ABB RAPID module: Module1.mod

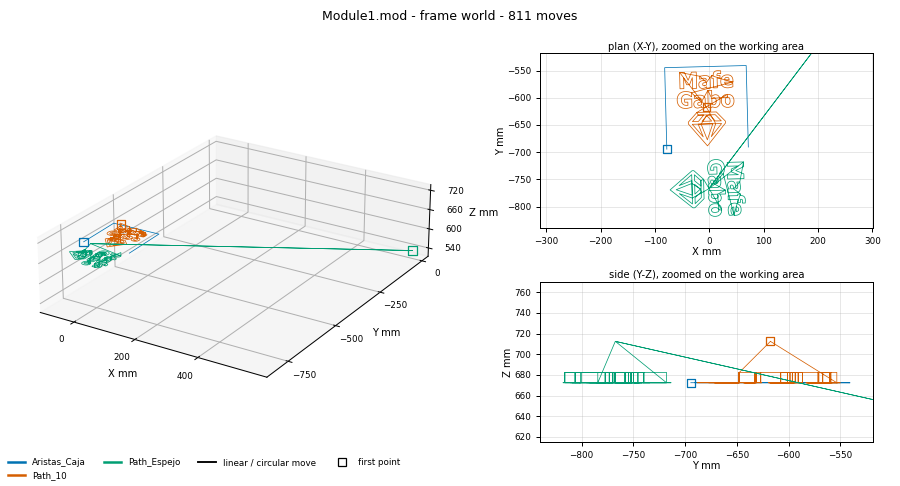
[picture p0: tool path of Module1.mod in frame world, 811 of 815 moves have a stored position in this frame; points joined in program order, loops and branches not executed]
MODULE Module1
	TASK PERS tooldata Marcador_TCP:=[TRUE,[[84.5459,-0.173285,134.639],[1,0,0,0]],[1,[1,2,3],[1,0,0,0],0,0,0]];
    !TASK PERS tooldata wcaja:=[FALSE,TRUE,"",[[-78.3768,-694.538,672.47],[0.999913,-0.00011372,0.00016022,0.0132033]],[[-74.9038,-552.314,679.445],[0.0262226,-0.999656,6.92619E-06,1.8063E-05]]];
    !TASK PERS wobjdata Caja:=[FALSE,TRUE,"",[[-250,0,346],[1,0,0,0]],[[750,75,154],[0.707106781,0,0,-0.707106781]]];
    !TASK PERS wobjdata Caja:=[FALSE,TRUE,"",[[-78.3768,-694.538,672.47],[0.999913,-0.00011372,0.00016022,0.0132033]],[[-74.9038,-552.314,679.445],[0.0262226,-0.999656,0.000006926,0.000018063]]];
    !TASK PERS wobjdata wcaja:=[FALSE,TRUE,"",[[-78.3768,-694.538,672.47],[0.999913,-0.00011372,0.00016022,0.0132033]],[[-74.9038,-552.314,679.445],[0.0262226,-0.999656,6.92619E-06,1.8063E-05]]];
    CONST robtarget Home:=[[75.173285,80.619495586,38.961602814],[0.353553391,-0.612372436,0.612372436,0.353553391],[0,0,0,0],[9E+09,9E+09,9E+09,9E+09,9E+09,9E+09]];
    CONST robtarget Target_10:=[[0,0,0],[0.353553391,0.612372436,0.612372436,-0.353553391],[0,-1,0,0],[9E+09,9E+09,9E+09,9E+09,9E+09,9E+09]];
    CONST robtarget Target_20:=[[0,150,0],[0.353553391,0.612372436,0.612372436,-0.353553391],[0,-1,0,0],[9E+09,9E+09,9E+09,9E+09,9E+09,9E+09]];
    CONST robtarget Target_30:=[[150,150,0],[0.353553391,0.612372436,0.612372436,-0.353553391],[-1,0,-1,0],[9E+09,9E+09,9E+09,9E+09,9E+09,9E+09]];
    CONST robtarget Target_40:=[[150,0,0],[0.353553391,0.612372436,0.612372436,-0.353553391],[-1,0,-1,0],[9E+09,9E+09,9E+09,9E+09,9E+09,9E+09]];
    CONST robtarget Target_50:=[[27.192,140.456999999,10],[0,0.866025404,0,-0.499999999],[0,0,0,0],[9E+09,9E+09,9E+09,9E+09,9E+09,9E+09]];
    CONST robtarget Target_60:=[[27.192,140.457,0],[0.353553391,0.612372436,0.612372436,-0.353553391],[-2,0,-1,0],[9E+09,9E+09,9E+09,9E+09,9E+09,9E+09]];
    CONST robtarget Target_70:=[[35.871,140.457,0],[0.353553391,0.612372436,0.612372436,-0.353553391],[-2,0,-1,0],[9E+09,9E+09,9E+09,9E+09,9E+09,9E+09]];
    CONST robtarget Target_80:=[[42.532,125.651,0],[0.353553391,0.612372436,0.612372436,-0.353553391],[-2,0,-1,0],[9E+09,9E+09,9E+09,9E+09,9E+09,9E+09]];
    CONST robtarget Target_90:=[[49.145,140.457,0],[0.353553391,0.612372436,0.612372436,-0.353553391],[-2,0,-1,0],[9E+09,9E+09,9E+09,9E+09,9E+09,9E+09]];
    CONST robtarget Target_100:=[[57.824,140.457,0],[0.353553391,0.612372436,0.612372436,-0.353553391],[-2,0,-1,0],[9E+09,9E+09,9E+09,9E+09,9E+09,9E+09]];
    CONST robtarget Target_110:=[[57.824,110.457,0],[0.353553391,0.612372436,0.612372436,-0.353553391],[-2,0,-1,0],[9E+09,9E+09,9E+09,9E+09,9E+09,9E+09]];
    CONST robtarget Target_120:=[[50.336,110.457,0],[0.353553391,0.612372436,0.612372436,-0.353553391],[-2,0,-1,0],[9E+09,9E+09,9E+09,9E+09,9E+09,9E+09]];
    CONST robtarget Target_130:=[[50.336,130.343,0],[0.353553391,0.612372436,0.612372436,-0.353553391],[-2,0,-1,0],[9E+09,9E+09,9E+09,9E+09,9E+09,9E+09]];
    CONST robtarget Target_140:=[[44.891,117.507,0],[0.353553391,0.612372436,0.612372436,-0.353553391],[-2,0,-1,0],[9E+09,9E+09,9E+09,9E+09,9E+09,9E+09]];
    CONST robtarget Target_150:=[[39.737,117.507,0],[0.353553391,0.612372436,0.612372436,-0.353553391],[-2,0,-1,0],[9E+09,9E+09,9E+09,9E+09,9E+09,9E+09]];
    CONST robtarget Target_160:=[[34.291,130.343,0],[0.353553391,0.612372436,0.612372436,-0.353553391],[-2,0,-1,0],[9E+09,9E+09,9E+09,9E+09,9E+09,9E+09]];
    CONST robtarget Target_170:=[[34.291,110.457,0],[0.353553391,0.612372436,0.612372436,-0.353553391],[-2,0,-1,0],[9E+09,9E+09,9E+09,9E+09,9E+09,9E+09]];
    CONST robtarget Target_180:=[[27.192,110.457,0],[0.353553391,0.612372436,0.612372436,-0.353553391],[-2,0,-1,0],[9E+09,9E+09,9E+09,9E+09,9E+09,9E+09]];
    CONST robtarget Target_190:=[[27.192,140.457,0],[0.353553391,0.612372436,0.612372436,-0.353553391],[-2,0,-1,0],[9E+09,9E+09,9E+09,9E+09,9E+09,9E+09]];
    CONST robtarget Target_200:=[[27.192,140.457,10],[0.353553391,0.612372436,0.612372436,-0.353553391],[-2,0,-1,0],[9E+09,9E+09,9E+09,9E+09,9E+09,9E+09]];
    CONST robtarget Target_210:=[[63.829,132.604,10],[0.353553391,0.612372436,0.612372436,-0.353553391],[-2,0,-1,0],[9E+09,9E+09,9E+09,9E+09,9E+09,9E+09]];
    CONST robtarget Target_220:=[[63.829,132.604,0],[0.353553391,0.612372436,0.612372436,-0.353553391],[-2,0,-1,0],[9E+09,9E+09,9E+09,9E+09,9E+09,9E+09]];
    CONST robtarget Target_230:=[[71.925,133.722,0],[0.353553391,0.612372436,0.612372436,-0.353553391],[-2,0,-1,0],[9E+09,9E+09,9E+09,9E+09,9E+09,9E+09]];
    CONST robtarget Target_240:=[[73.075,133.702,0],[0.353553391,0.612372436,0.612372436,-0.353553391],[-2,0,-1,0],[9E+09,9E+09,9E+09,9E+09,9E+09,9E+09]];
    CONST robtarget Target_250:=[[74.399,133.623,0],[0.353553391,0.612372436,0.612372436,-0.353553391],[-2,0,-1,0],[9E+09,9E+09,9E+09,9E+09,9E+09,9E+09]];
    CONST robtarget Target_260:=[[76.16,133.399,0],[0.353553391,0.612372436,0.612372436,-0.353553391],[-2,0,-1,0],[9E+09,9E+09,9E+09,9E+09,9E+09,9E+09]];
    CONST robtarget Target_270:=[[77.475,133.111,0],[0.353553391,0.612372436,0.612372436,-0.353553391],[-2,0,-1,0],[9E+09,9E+09,9E+09,9E+09,9E+09,9E+09]];
    CONST robtarget Target_280:=[[78.922,132.618,0],[0.353553391,0.612372436,0.612372436,-0.353553391],[-2,0,-1,0],[9E+09,9E+09,9E+09,9E+09,9E+09,9E+09]];
    CONST robtarget Target_290:=[[80.057,132.032,0],[0.353553391,0.612372436,0.612372436,-0.353553391],[-2,0,-1,0],[9E+09,9E+09,9E+09,9E+09,9E+09,9E+09]];
    CONST robtarget Target_300:=[[81.155,131.169,0],[0.353553391,0.612372436,0.612372436,-0.353553391],[-2,0,-1,0],[9E+09,9E+09,9E+09,9E+09,9E+09,9E+09]];
    CONST robtarget Target_310:=[[81.768,130.466,0],[0.353553391,0.612372436,0.612372436,-0.353553391],[-2,0,-1,0],[9E+09,9E+09,9E+09,9E+09,9E+09,9E+09]];
    CONST robtarget Target_320:=[[82.441,129.318,0],[0.353553391,0.612372436,0.612372436,-0.353553391],[-2,0,-1,0],[9E+09,9E+09,9E+09,9E+09,9E+09,9E+09]];
    CONST robtarget Target_330:=[[82.754,128.475,0],[0.353553391,0.612372436,0.612372436,-0.353553391],[-2,0,-1,0],[9E+09,9E+09,9E+09,9E+09,9E+09,9E+09]];
    CONST robtarget Target_340:=[[82.989,127.436,0],[0.353553391,0.612372436,0.612372436,-0.353553391],[-2,0,-1,0],[9E+09,9E+09,9E+09,9E+09,9E+09,9E+09]];
    CONST robtarget Target_350:=[[83.108,125.846,0],[0.353553391,0.612372436,0.612372436,-0.353553391],[-2,0,-1,0],[9E+09,9E+09,9E+09,9E+09,9E+09,9E+09]];
    CONST robtarget Target_360:=[[83.108,110.457,0],[0.353553391,0.612372436,0.612372436,-0.353553391],[-2,0,-1,0],[9E+09,9E+09,9E+09,9E+09,9E+09,9E+09]];
    CONST robtarget Target_370:=[[76.106,110.457,0],[0.353553391,0.612372436,0.612372436,-0.353553391],[-2,0,-1,0],[9E+09,9E+09,9E+09,9E+09,9E+09,9E+09]];
    CONST robtarget Target_380:=[[76.106,112.863,0],[0.353553391,0.612372436,0.612372436,-0.353553391],[-2,0,-1,0],[9E+09,9E+09,9E+09,9E+09,9E+09,9E+09]];
    CONST robtarget Target_390:=[[73.262,110.797,0],[0.353553391,0.612372436,0.612372436,-0.353553391],[-2,0,-1,0],[9E+09,9E+09,9E+09,9E+09,9E+09,9E+09]];
    CONST robtarget Target_400:=[[68.91,109.849,0],[0.353553391,0.612372436,0.612372436,-0.353553391],[-2,0,-1,0],[9E+09,9E+09,9E+09,9E+09,9E+09,9E+09]];
    CONST robtarget Target_410:=[[67.809,109.921,0],[0.353553391,0.612372436,0.612372436,-0.353553391],[-2,0,-1,0],[9E+09,9E+09,9E+09,9E+09,9E+09,9E+09]];
    CONST robtarget Target_420:=[[66.698,110.161,0],[0.353553391,0.612372436,0.612372436,-0.353553391],[-2,0,-1,0],[9E+09,9E+09,9E+09,9E+09,9E+09,9E+09]];
    CONST robtarget Target_430:=[[65.802,110.508,0],[0.353553391,0.612372436,0.612372436,-0.353553391],[-2,0,-1,0],[9E+09,9E+09,9E+09,9E+09,9E+09,9E+09]];
    CONST robtarget Target_440:=[[64.811,111.094,0],[0.353553391,0.612372436,0.612372436,-0.353553391],[-2,0,-1,0],[9E+09,9E+09,9E+09,9E+09,9E+09,9E+09]];
    CONST robtarget Target_450:=[[63.886,111.896,0],[0.353553391,0.612372436,0.612372436,-0.353553391],[-2,0,-1,0],[9E+09,9E+09,9E+09,9E+09,9E+09,9E+09]];
    CONST robtarget Target_460:=[[63.01,112.999,0],[0.353553391,0.612372436,0.612372436,-0.353553391],[-2,0,-1,0],[9E+09,9E+09,9E+09,9E+09,9E+09,9E+09]];
    CONST robtarget Target_470:=[[62.505,113.958,0],[0.353553391,0.612372436,0.612372436,-0.353553391],[-2,0,-1,0],[9E+09,9E+09,9E+09,9E+09,9E+09,9E+09]];
    CONST robtarget Target_480:=[[62.106,115.23,0],[0.353553391,0.612372436,0.612372436,-0.353553391],[-2,0,-1,0],[9E+09,9E+09,9E+09,9E+09,9E+09,9E+09]];
    CONST robtarget Target_490:=[[61.935,116.747,0],[0.353553391,0.612372436,0.612372436,-0.353553391],[-2,0,-1,0],[9E+09,9E+09,9E+09,9E+09,9E+09,9E+09]];
    CONST robtarget Target_500:=[[61.956,117.693,0],[0.353553391,0.612372436,0.612372436,-0.353553391],[-2,0,-1,0],[9E+09,9E+09,9E+09,9E+09,9E+09,9E+09]];
    CONST robtarget Target_510:=[[62.24,119.422,0],[0.353553391,0.612372436,0.612372436,-0.353553391],[-2,0,-1,0],[9E+09,9E+09,9E+09,9E+09,9E+09,9E+09]];
    CONST robtarget Target_520:=[[62.681,120.558,0],[0.353553391,0.612372436,0.612372436,-0.353553391],[-2,0,-1,0],[9E+09,9E+09,9E+09,9E+09,9E+09,9E+09]];
    CONST robtarget Target_530:=[[63.326,121.537,0],[0.353553391,0.612372436,0.612372436,-0.353553391],[-2,0,-1,0],[9E+09,9E+09,9E+09,9E+09,9E+09,9E+09]];
    CONST robtarget Target_540:=[[64.156,122.386,0],[0.353553391,0.612372436,0.612372436,-0.353553391],[-2,0,-1,0],[9E+09,9E+09,9E+09,9E+09,9E+09,9E+09]];
    CONST robtarget Target_550:=[[65.088,123.055,0],[0.353553391,0.612372436,0.612372436,-0.353553391],[-2,0,-1,0],[9E+09,9E+09,9E+09,9E+09,9E+09,9E+09]];
    CONST robtarget Target_560:=[[65.847,123.463,0],[0.353553391,0.612372436,0.612372436,-0.353553391],[-2,0,-1,0],[9E+09,9E+09,9E+09,9E+09,9E+09,9E+09]];
    CONST robtarget Target_570:=[[69.214,124.548,0],[0.353553391,0.612372436,0.612372436,-0.353553391],[-2,0,-1,0],[9E+09,9E+09,9E+09,9E+09,9E+09,9E+09]];
    CONST robtarget Target_580:=[[70.751,124.795,0],[0.353553391,0.612372436,0.612372436,-0.353553391],[-2,0,-1,0],[9E+09,9E+09,9E+09,9E+09,9E+09,9E+09]];
    CONST robtarget Target_590:=[[72.603,125.014,0],[0.353553391,0.612372436,0.612372436,-0.353553391],[-2,0,-1,0],[9E+09,9E+09,9E+09,9E+09,9E+09,9E+09]];
    CONST robtarget Target_600:=[[74.414,125.184,0],[0.353553391,0.612372436,0.612372436,-0.353553391],[-2,0,-1,0],[9E+09,9E+09,9E+09,9E+09,9E+09,9E+09]];
    CONST robtarget Target_610:=[[76.155,125.311,0],[0.353553391,0.612372436,0.612372436,-0.353553391],[-2,0,-1,0],[9E+09,9E+09,9E+09,9E+09,9E+09,9E+09]];
    CONST robtarget Target_620:=[[76.155,125.432,0],[0.353553391,0.612372436,0.612372436,-0.353553391],[-2,0,-1,0],[9E+09,9E+09,9E+09,9E+09,9E+09,9E+09]];
    CONST robtarget Target_630:=[[76.114,126.039,0],[0.353553391,0.612372436,0.612372436,-0.353553391],[-2,0,-1,0],[9E+09,9E+09,9E+09,9E+09,9E+09,9E+09]];
    CONST robtarget Target_640:=[[75.849,126.936,0],[0.353553391,0.612372436,0.612372436,-0.353553391],[-2,0,-1,0],[9E+09,9E+09,9E+09,9E+09,9E+09,9E+09]];
    CONST robtarget Target_650:=[[75.219,127.729,0],[0.353553391,0.612372436,0.612372436,-0.353553391],[-2,0,-1,0],[9E+09,9E+09,9E+09,9E+09,9E+09,9E+09]];
    CONST robtarget Target_660:=[[74.486,128.154,0],[0.353553391,0.612372436,0.612372436,-0.353553391],[-2,0,-1,0],[9E+09,9E+09,9E+09,9E+09,9E+09,9E+09]];
    CONST robtarget Target_670:=[[73.351,128.499,0],[0.353553391,0.612372436,0.612372436,-0.353553391],[-2,0,-1,0],[9E+09,9E+09,9E+09,9E+09,9E+09,9E+09]];
    CONST robtarget Target_680:=[[72.285,128.661,0],[0.353553391,0.612372436,0.612372436,-0.353553391],[-2,0,-1,0],[9E+09,9E+09,9E+09,9E+09,9E+09,9E+09]];
    CONST robtarget Target_690:=[[71.471,128.72,0],[0.353553391,0.612372436,0.612372436,-0.353553391],[-2,0,-1,0],[9E+09,9E+09,9E+09,9E+09,9E+09,9E+09]];
    CONST robtarget Target_700:=[[70.612,128.739,0],[0.353553391,0.612372436,0.612372436,-0.353553391],[-2,0,-1,0],[9E+09,9E+09,9E+09,9E+09,9E+09,9E+09]];
    CONST robtarget Target_710:=[[64.437,127.134,0],[0.353553391,0.612372436,0.612372436,-0.353553391],[-2,0,-1,0],[9E+09,9E+09,9E+09,9E+09,9E+09,9E+09]];
    CONST robtarget Target_720:=[[63.829,127.134,0],[0.353553391,0.612372436,0.612372436,-0.353553391],[-2,0,-1,0],[9E+09,9E+09,9E+09,9E+09,9E+09,9E+09]];
    CONST robtarget Target_730:=[[63.829,132.604,0],[0.353553391,0.612372436,0.612372436,-0.353553391],[-2,0,-1,0],[9E+09,9E+09,9E+09,9E+09,9E+09,9E+09]];
    CONST robtarget Target_740:=[[63.829,132.604,10],[0.353553391,0.612372436,0.612372436,-0.353553391],[-2,0,-1,0],[9E+09,9E+09,9E+09,9E+09,9E+09,9E+09]];
    CONST robtarget Target_750:=[[76.106,121.056,10],[0.353553391,0.612372436,0.612372436,-0.353553391],[-2,0,-1,0],[9E+09,9E+09,9E+09,9E+09,9E+09,9E+09]];
    CONST robtarget Target_760:=[[76.106,121.056,0],[0.353553391,0.612372436,0.612372436,-0.353553391],[-2,0,-1,0],[9E+09,9E+09,9E+09,9E+09,9E+09,9E+09]];
    CONST robtarget Target_770:=[[71.025,120.23,0],[0.353553391,0.612372436,0.612372436,-0.353553391],[-2,0,-1,0],[9E+09,9E+09,9E+09,9E+09,9E+09,9E+09]];
    CONST robtarget Target_780:=[[70.06,119.739,0],[0.353553391,0.612372436,0.612372436,-0.353553391],[-2,0,-1,0],[9E+09,9E+09,9E+09,9E+09,9E+09,9E+09]];
    CONST robtarget Target_790:=[[69.338,118.892,0],[0.353553391,0.612372436,0.612372436,-0.353553391],[-2,0,-1,0],[9E+09,9E+09,9E+09,9E+09,9E+09,9E+09]];
    CONST robtarget Target_800:=[[69.114,118.205,0],[0.353553391,0.612372436,0.612372436,-0.353553391],[-2,0,-1,0],[9E+09,9E+09,9E+09,9E+09,9E+09,9E+09]];
    CONST robtarget Target_810:=[[69.056,117.55,0],[0.353553391,0.612372436,0.612372436,-0.353553391],[-2,0,-1,0],[9E+09,9E+09,9E+09,9E+09,9E+09,9E+09]];
    CONST robtarget Target_820:=[[69.091,116.93,0],[0.353553391,0.612372436,0.612372436,-0.353553391],[-2,0,-1,0],[9E+09,9E+09,9E+09,9E+09,9E+09,9E+09]];
    CONST robtarget Target_830:=[[69.292,116.148,0],[0.353553391,0.612372436,0.612372436,-0.353553391],[-2,0,-1,0],[9E+09,9E+09,9E+09,9E+09,9E+09,9E+09]];
    CONST robtarget Target_840:=[[69.919,115.356,0],[0.353553391,0.612372436,0.612372436,-0.353553391],[-2,0,-1,0],[9E+09,9E+09,9E+09,9E+09,9E+09,9E+09]];
    CONST robtarget Target_850:=[[70.774,114.964,0],[0.353553391,0.612372436,0.612372436,-0.353553391],[-2,0,-1,0],[9E+09,9E+09,9E+09,9E+09,9E+09,9E+09]];
    CONST robtarget Target_860:=[[71.742,114.79,0],[0.353553391,0.612372436,0.612372436,-0.353553391],[-2,0,-1,0],[9E+09,9E+09,9E+09,9E+09,9E+09,9E+09]];
    CONST robtarget Target_870:=[[72.46,114.76,0],[0.353553391,0.612372436,0.612372436,-0.353553391],[-2,0,-1,0],[9E+09,9E+09,9E+09,9E+09,9E+09,9E+09]];
    CONST robtarget Target_880:=[[72.459,114.76,0],[0.353553391,0.612372436,0.612372436,-0.353553391],[-2,0,-1,0],[9E+09,9E+09,9E+09,9E+09,9E+09,9E+09]];
    CONST robtarget Target_890:=[[73.597,114.916,0],[0.353553391,0.612372436,0.612372436,-0.353553391],[-2,0,-1,0],[9E+09,9E+09,9E+09,9E+09,9E+09,9E+09]];
    CONST robtarget Target_900:=[[74.622,115.309,0],[0.353553391,0.612372436,0.612372436,-0.353553391],[-2,0,-1,0],[9E+09,9E+09,9E+09,9E+09,9E+09,9E+09]];
    CONST robtarget Target_910:=[[75.105,115.58,0],[0.353553391,0.612372436,0.612372436,-0.353553391],[-2,0,-1,0],[9E+09,9E+09,9E+09,9E+09,9E+09,9E+09]];
    CONST robtarget Target_920:=[[75.771,116.063,0],[0.353553391,0.612372436,0.612372436,-0.353553391],[-2,0,-1,0],[9E+09,9E+09,9E+09,9E+09,9E+09,9E+09]];
    CONST robtarget Target_930:=[[76.106,116.364,0],[0.353553391,0.612372436,0.612372436,-0.353553391],[-2,0,-1,0],[9E+09,9E+09,9E+09,9E+09,9E+09,9E+09]];
    CONST robtarget Target_940:=[[76.106,121.056,0],[0.353553391,0.612372436,0.612372436,-0.353553391],[-2,0,-1,0],[9E+09,9E+09,9E+09,9E+09,9E+09,9E+09]];
    CONST robtarget Target_950:=[[76.106,121.056,10],[0.353553391,0.612372436,0.612372436,-0.353553391],[-2,0,-1,0],[9E+09,9E+09,9E+09,9E+09,9E+09,9E+09]];
    CONST robtarget Target_960:=[[86.049,133.09,10],[0.353553391,0.612372436,0.612372436,-0.353553391],[-1,0,-1,0],[9E+09,9E+09,9E+09,9E+09,9E+09,9E+09]];
    CONST robtarget Target_970:=[[86.049,133.09,0],[0.353553391,0.612372436,0.612372436,-0.353553391],[-1,0,-1,0],[9E+09,9E+09,9E+09,9E+09,9E+09,9E+09]];
    CONST robtarget Target_980:=[[88.87,133.09,0],[0.353553391,0.612372436,0.612372436,-0.353553391],[-1,0,-1,0],[9E+09,9E+09,9E+09,9E+09,9E+09,9E+09]];
    CONST robtarget Target_990:=[[88.87,133.722,0],[0.353553391,0.612372436,0.612372436,-0.353553391],[-1,0,-1,0],[9E+09,9E+09,9E+09,9E+09,9E+09,9E+09]];
    CONST robtarget Target_1000:=[[88.943,135.17,0],[0.353553391,0.612372436,0.612372436,-0.353553391],[-1,0,-1,0],[9E+09,9E+09,9E+09,9E+09,9E+09,9E+09]];
    CONST robtarget Target_1010:=[[89.33,137.086,0],[0.353553391,0.612372436,0.612372436,-0.353553391],[-1,0,-1,0],[9E+09,9E+09,9E+09,9E+09,9E+09,9E+09]];
    CONST robtarget Target_1020:=[[90.035,138.666,0],[0.353553391,0.612372436,0.612372436,-0.353553391],[-1,0,-1,0],[9E+09,9E+09,9E+09,9E+09,9E+09,9E+09]];
    CONST robtarget Target_1030:=[[90.843,139.72,0],[0.353553391,0.612372436,0.612372436,-0.353553391],[-1,0,-1,0],[9E+09,9E+09,9E+09,9E+09,9E+09,9E+09]];
    CONST robtarget Target_1040:=[[92.423,140.908,0],[0.353553391,0.612372436,0.612372436,-0.353553391],[-1,0,-1,0],[9E+09,9E+09,9E+09,9E+09,9E+09,9E+09]];
    CONST robtarget Target_1050:=[[94.644,141.698,0],[0.353553391,0.612372436,0.612372436,-0.353553391],[-1,0,-1,0],[9E+09,9E+09,9E+09,9E+09,9E+09,9E+09]];
    CONST robtarget Target_1060:=[[96.483,141.95,0],[0.353553391,0.612372436,0.612372436,-0.353553391],[-1,-1,-1,0],[9E+09,9E+09,9E+09,9E+09,9E+09,9E+09]];
    CONST robtarget Target_1070:=[[97.646,141.988,0],[0.353553391,0.612372436,0.612372436,-0.353553391],[-1,-1,0,0],[9E+09,9E+09,9E+09,9E+09,9E+09,9E+09]];
    CONST robtarget Target_1080:=[[102.8,141.575,0],[0.353553391,0.612372436,0.612372436,-0.353553391],[-1,-1,0,0],[9E+09,9E+09,9E+09,9E+09,9E+09,9E+09]];
    CONST robtarget Target_1090:=[[102.8,136.47,0],[0.353553391,0.612372436,0.612372436,-0.353553391],[-1,-1,0,0],[9E+09,9E+09,9E+09,9E+09,9E+09,9E+09]];
    CONST robtarget Target_1100:=[[102.265,136.47,0],[0.353553391,0.612372436,0.612372436,-0.353553391],[-1,-1,0,0],[9E+09,9E+09,9E+09,9E+09,9E+09,9E+09]];
    CONST robtarget Target_1110:=[[99.372,136.98,0],[0.353553391,0.612372436,0.612372436,-0.353553391],[-1,-1,0,0],[9E+09,9E+09,9E+09,9E+09,9E+09,9E+09]];
    CONST robtarget Target_1120:=[[98.552,136.947,0],[0.353553391,0.612372436,0.612372436,-0.353553391],[-1,-1,0,0],[9E+09,9E+09,9E+09,9E+09,9E+09,9E+09]];
    CONST robtarget Target_1130:=[[97.623,136.799,0],[0.353553391,0.612372436,0.612372436,-0.353553391],[-1,-1,0,0],[9E+09,9E+09,9E+09,9E+09,9E+09,9E+09]];
    CONST robtarget Target_1140:=[[96.675,136.388,0],[0.353553391,0.612372436,0.612372436,-0.353553391],[-1,-1,0,0],[9E+09,9E+09,9E+09,9E+09,9E+09,9E+09]];
    CONST robtarget Target_1150:=[[96.077,135.652,0],[0.353553391,0.612372436,0.612372436,-0.353553391],[-1,0,-1,0],[9E+09,9E+09,9E+09,9E+09,9E+09,9E+09]];
    CONST robtarget Target_1160:=[[95.864,135.05,0],[0.353553391,0.612372436,0.612372436,-0.353553391],[-1,0,-1,0],[9E+09,9E+09,9E+09,9E+09,9E+09,9E+09]];
    CONST robtarget Target_1170:=[[95.723,134.236,0],[0.353553391,0.612372436,0.612372436,-0.353553391],[-1,0,-1,0],[9E+09,9E+09,9E+09,9E+09,9E+09,9E+09]];
    CONST robtarget Target_1180:=[[95.677,133.26,0],[0.353553391,0.612372436,0.612372436,-0.353553391],[-1,0,-1,0],[9E+09,9E+09,9E+09,9E+09,9E+09,9E+09]];
    CONST robtarget Target_1190:=[[95.677,133.09,0],[0.353553391,0.612372436,0.612372436,-0.353553391],[-1,0,-1,0],[9E+09,9E+09,9E+09,9E+09,9E+09,9E+09]];
    CONST robtarget Target_1200:=[[101.293,133.09,0],[0.353553391,0.612372436,0.612372436,-0.353553391],[-1,-1,0,0],[9E+09,9E+09,9E+09,9E+09,9E+09,9E+09]];
    CONST robtarget Target_1210:=[[101.293,128.179,0],[0.353553391,0.612372436,0.612372436,-0.353553391],[-1,-1,0,0],[9E+09,9E+09,9E+09,9E+09,9E+09,9E+09]];
    CONST robtarget Target_1220:=[[95.92,128.179,0],[0.353553391,0.612372436,0.612372436,-0.353553391],[-1,0,-1,0],[9E+09,9E+09,9E+09,9E+09,9E+09,9E+09]];
    CONST robtarget Target_1230:=[[95.92,110.457,0],[0.353553391,0.612372436,0.612372436,-0.353553391],[-1,0,-1,0],[9E+09,9E+09,9E+09,9E+09,9E+09,9E+09]];
    CONST robtarget Target_1240:=[[88.87,110.457,0],[0.353553391,0.612372436,0.612372436,-0.353553391],[-1,0,-1,0],[9E+09,9E+09,9E+09,9E+09,9E+09,9E+09]];
    CONST robtarget Target_1250:=[[88.87,128.179,0],[0.353553391,0.612372436,0.612372436,-0.353553391],[-1,0,-1,0],[9E+09,9E+09,9E+09,9E+09,9E+09,9E+09]];
    CONST robtarget Target_1260:=[[86.049,128.179,0],[0.353553391,0.612372436,0.612372436,-0.353553391],[-1,0,-1,0],[9E+09,9E+09,9E+09,9E+09,9E+09,9E+09]];
    CONST robtarget Target_1270:=[[86.049,133.09,0],[0.353553391,0.612372436,0.612372436,-0.353553391],[-1,0,-1,0],[9E+09,9E+09,9E+09,9E+09,9E+09,9E+09]];
    CONST robtarget Target_1280:=[[86.049,133.09,10],[0.353553391,0.612372436,0.612372436,-0.353553391],[-1,0,-1,0],[9E+09,9E+09,9E+09,9E+09,9E+09,9E+09]];
    CONST robtarget Target_1290:=[[109.485,124.679,10],[0.353553391,0.612372436,0.612372436,-0.353553391],[-1,-1,0,0],[9E+09,9E+09,9E+09,9E+09,9E+09,9E+09]];
    CONST robtarget Target_1300:=[[109.485,124.679,0],[0.353553391,0.612372436,0.612372436,-0.353553391],[-1,-1,0,0],[9E+09,9E+09,9E+09,9E+09,9E+09,9E+09]];
    CONST robtarget Target_1310:=[[109.701,126.061,0],[0.353553391,0.612372436,0.612372436,-0.353553391],[-1,-1,0,0],[9E+09,9E+09,9E+09,9E+09,9E+09,9E+09]];
    CONST robtarget Target_1320:=[[110.324,127.465,0],[0.353553391,0.612372436,0.612372436,-0.353553391],[-1,-1,0,0],[9E+09,9E+09,9E+09,9E+09,9E+09,9E+09]];
    CONST robtarget Target_1330:=[[111.27,128.475,0],[0.353553391,0.612372436,0.612372436,-0.353553391],[-1,-1,0,0],[9E+09,9E+09,9E+09,9E+09,9E+09,9E+09]];
    CONST robtarget Target_1340:=[[112.867,129.166,0],[0.353553391,0.612372436,0.612372436,-0.353553391],[-1,-1,0,0],[9E+09,9E+09,9E+09,9E+09,9E+09,9E+09]];
    CONST robtarget Target_1350:=[[114.033,129.273,0],[0.353553391,0.612372436,0.612372436,-0.353553391],[-1,-1,0,0],[9E+09,9E+09,9E+09,9E+09,9E+09,9E+09]];
    CONST robtarget Target_1360:=[[114.895,129.209,0],[0.353553391,0.612372436,0.612372436,-0.353553391],[-1,-1,0,0],[9E+09,9E+09,9E+09,9E+09,9E+09,9E+09]];
    CONST robtarget Target_1370:=[[116.013,128.871,0],[0.353553391,0.612372436,0.612372436,-0.353553391],[-1,-1,0,0],[9E+09,9E+09,9E+09,9E+09,9E+09,9E+09]];
    CONST robtarget Target_1380:=[[116.864,128.257,0],[0.353553391,0.612372436,0.612372436,-0.353553391],[-1,-1,0,0],[9E+09,9E+09,9E+09,9E+09,9E+09,9E+09]];
    CONST robtarget Target_1390:=[[117.585,127.137,0],[0.353553391,0.612372436,0.612372436,-0.353553391],[-1,-1,0,0],[9E+09,9E+09,9E+09,9E+09,9E+09,9E+09]];
    CONST robtarget Target_1400:=[[117.862,126.264,0],[0.353553391,0.612372436,0.612372436,-0.353553391],[-1,-1,0,0],[9E+09,9E+09,9E+09,9E+09,9E+09,9E+09]];
    CONST robtarget Target_1410:=[[118,125.407,0],[0.353553391,0.612372436,0.612372436,-0.353553391],[-1,-1,0,0],[9E+09,9E+09,9E+09,9E+09,9E+09,9E+09]];
    CONST robtarget Target_1420:=[[118.043,124.679,0],[0.353553391,0.612372436,0.612372436,-0.353553391],[-1,-1,0,0],[9E+09,9E+09,9E+09,9E+09,9E+09,9E+09]];
    CONST robtarget Target_1430:=[[109.485,124.679,0],[0.353553391,0.612372436,0.612372436,-0.353553391],[-1,-1,0,0],[9E+09,9E+09,9E+09,9E+09,9E+09,9E+09]];
    CONST robtarget Target_1440:=[[109.485,124.679,10],[0.353553391,0.612372436,0.612372436,-0.353553391],[-1,-1,0,0],[9E+09,9E+09,9E+09,9E+09,9E+09,9E+09]];
    CONST robtarget Target_1450:=[[124.996,120.424,10],[0.353553391,0.612372436,0.612372436,-0.353553391],[-1,-1,0,0],[9E+09,9E+09,9E+09,9E+09,9E+09,9E+09]];
    CONST robtarget Target_1460:=[[124.996,120.424,0],[0.353553391,0.612372436,0.612372436,-0.353553391],[-1,-1,0,0],[9E+09,9E+09,9E+09,9E+09,9E+09,9E+09]];
    CONST robtarget Target_1470:=[[109.51,120.424,0],[0.353553391,0.612372436,0.612372436,-0.353553391],[-1,-1,0,0],[9E+09,9E+09,9E+09,9E+09,9E+09,9E+09]];
    CONST robtarget Target_1480:=[[110.356,117.497,0],[0.353553391,0.612372436,0.612372436,-0.353553391],[-1,-1,0,0],[9E+09,9E+09,9E+09,9E+09,9E+09,9E+09]];
    CONST robtarget Target_1490:=[[111.754,116.065,0],[0.353553391,0.612372436,0.612372436,-0.353553391],[-1,-1,0,0],[9E+09,9E+09,9E+09,9E+09,9E+09,9E+09]];
    CONST robtarget Target_1500:=[[113.375,115.326,0],[0.353553391,0.612372436,0.612372436,-0.353553391],[-1,-1,0,0],[9E+09,9E+09,9E+09,9E+09,9E+09,9E+09]];
    CONST robtarget Target_1510:=[[115.333,114.996,0],[0.353553391,0.612372436,0.612372436,-0.353553391],[-1,-1,0,0],[9E+09,9E+09,9E+09,9E+09,9E+09,9E+09]];
    CONST robtarget Target_1520:=[[117.175,114.979,0],[0.353553391,0.612372436,0.612372436,-0.353553391],[-1,-1,0,0],[9E+09,9E+09,9E+09,9E+09,9E+09,9E+09]];
    CONST robtarget Target_1530:=[[118.717,115.194,0],[0.353553391,0.612372436,0.612372436,-0.353553391],[-1,-1,0,0],[9E+09,9E+09,9E+09,9E+09,9E+09,9E+09]];
    CONST robtarget Target_1540:=[[120.709,115.808,0],[0.353553391,0.612372436,0.612372436,-0.353553391],[-1,-1,0,0],[9E+09,9E+09,9E+09,9E+09,9E+09,9E+09]];
    CONST robtarget Target_1550:=[[121.033,115.951,0],[0.353553391,0.612372436,0.612372436,-0.353553391],[-1,-1,0,0],[9E+09,9E+09,9E+09,9E+09,9E+09,9E+09]];
    CONST robtarget Target_1560:=[[123.829,117.555,0],[0.353553391,0.612372436,0.612372436,-0.353553391],[-1,-1,0,0],[9E+09,9E+09,9E+09,9E+09,9E+09,9E+09]];
    CONST robtarget Target_1570:=[[124.583,117.555,0],[0.353553391,0.612372436,0.612372436,-0.353553391],[-1,-1,0,0],[9E+09,9E+09,9E+09,9E+09,9E+09,9E+09]];
    CONST robtarget Target_1580:=[[124.583,111.721,0],[0.353553391,0.612372436,0.612372436,-0.353553391],[-1,-1,0,0],[9E+09,9E+09,9E+09,9E+09,9E+09,9E+09]];
    CONST robtarget Target_1590:=[[121.033,110.505,0],[0.353553391,0.612372436,0.612372436,-0.353553391],[-1,-1,0,0],[9E+09,9E+09,9E+09,9E+09,9E+09,9E+09]];
    CONST robtarget Target_1600:=[[115.709,109.849,0],[0.353553391,0.612372436,0.612372436,-0.353553391],[-1,-1,0,0],[9E+09,9E+09,9E+09,9E+09,9E+09,9E+09]];
    CONST robtarget Target_1610:=[[113.106,109.988,0],[0.353553391,0.612372436,0.612372436,-0.353553391],[-1,-1,0,0],[9E+09,9E+09,9E+09,9E+09,9E+09,9E+09]];
    CONST robtarget Target_1620:=[[110.207,110.564,0],[0.353553391,0.612372436,0.612372436,-0.353553391],[-1,-1,0,0],[9E+09,9E+09,9E+09,9E+09,9E+09,9E+09]];
    CONST robtarget Target_1630:=[[108.088,111.404,0],[0.353553391,0.612372436,0.612372436,-0.353553391],[-1,-1,0,0],[9E+09,9E+09,9E+09,9E+09,9E+09,9E+09]];
    CONST robtarget Target_1640:=[[106.39,112.481,0],[0.353553391,0.612372436,0.612372436,-0.353553391],[-1,-1,0,0],[9E+09,9E+09,9E+09,9E+09,9E+09,9E+09]];
    CONST robtarget Target_1650:=[[105.004,113.799,0],[0.353553391,0.612372436,0.612372436,-0.353553391],[-1,-1,0,0],[9E+09,9E+09,9E+09,9E+09,9E+09,9E+09]];
    CONST robtarget Target_1660:=[[103.854,115.462,0],[0.353553391,0.612372436,0.612372436,-0.353553391],[-1,-1,0,0],[9E+09,9E+09,9E+09,9E+09,9E+09,9E+09]];
    CONST robtarget Target_1670:=[[103.1,117.221,0],[0.353553391,0.612372436,0.612372436,-0.353553391],[-1,-1,0,0],[9E+09,9E+09,9E+09,9E+09,9E+09,9E+09]];
    CONST robtarget Target_1680:=[[102.678,118.94,0],[0.353553391,0.612372436,0.612372436,-0.353553391],[-1,-1,0,0],[9E+09,9E+09,9E+09,9E+09,9E+09,9E+09]];
    CONST robtarget Target_1690:=[[102.466,121.144,0],[0.353553391,0.612372436,0.612372436,-0.353553391],[-1,-1,0,0],[9E+09,9E+09,9E+09,9E+09,9E+09,9E+09]];
    CONST robtarget Target_1700:=[[102.503,122.901,0],[0.353553391,0.612372436,0.612372436,-0.353553391],[-1,-1,0,0],[9E+09,9E+09,9E+09,9E+09,9E+09,9E+09]];
    CONST robtarget Target_1710:=[[102.895,125.435,0],[0.353553391,0.612372436,0.612372436,-0.353553391],[-1,-1,0,0],[9E+09,9E+09,9E+09,9E+09,9E+09,9E+09]];
    CONST robtarget Target_1720:=[[103.544,127.348,0],[0.353553391,0.612372436,0.612372436,-0.353553391],[-1,-1,0,0],[9E+09,9E+09,9E+09,9E+09,9E+09,9E+09]];
    CONST robtarget Target_1730:=[[104.846,129.56,0],[0.353553391,0.612372436,0.612372436,-0.353553391],[-1,-1,0,0],[9E+09,9E+09,9E+09,9E+09,9E+09,9E+09]];
    CONST robtarget Target_1740:=[[107.173,131.787,0],[0.353553391,0.612372436,0.612372436,-0.353553391],[-1,-1,0,0],[9E+09,9E+09,9E+09,9E+09,9E+09,9E+09]];
    CONST robtarget Target_1750:=[[110.252,133.228,0],[0.353553391,0.612372436,0.612372436,-0.353553391],[-1,-1,0,0],[9E+09,9E+09,9E+09,9E+09,9E+09,9E+09]];
    CONST robtarget Target_1760:=[[112.653,133.696,0],[0.353553391,0.612372436,0.612372436,-0.353553391],[-1,-1,0,0],[9E+09,9E+09,9E+09,9E+09,9E+09,9E+09]];
    CONST robtarget Target_1770:=[[115.907,133.745,0],[0.353553391,0.612372436,0.612372436,-0.353553391],[-1,-1,0,0],[9E+09,9E+09,9E+09,9E+09,9E+09,9E+09]];
    CONST robtarget Target_1780:=[[118.059,133.408,0],[0.353553391,0.612372436,0.612372436,-0.353553391],[-1,-1,0,0],[9E+09,9E+09,9E+09,9E+09,9E+09,9E+09]];
    CONST robtarget Target_1790:=[[120.042,132.698,0],[0.353553391,0.612372436,0.612372436,-0.353553391],[-1,-1,0,0],[9E+09,9E+09,9E+09,9E+09,9E+09,9E+09]];
    CONST robtarget Target_1800:=[[121.361,131.894,0],[0.353553391,0.612372436,0.612372436,-0.353553391],[-1,-1,0,0],[9E+09,9E+09,9E+09,9E+09,9E+09,9E+09]];
    CONST robtarget Target_1810:=[[122.662,130.659,0],[0.353553391,0.612372436,0.612372436,-0.353553391],[-1,-1,0,0],[9E+09,9E+09,9E+09,9E+09,9E+09,9E+09]];
    CONST robtarget Target_1820:=[[123.82,128.868,0],[0.353553391,0.612372436,0.612372436,-0.353553391],[-1,-1,0,0],[9E+09,9E+09,9E+09,9E+09,9E+09,9E+09]];
    CONST robtarget Target_1830:=[[124.578,126.747,0],[0.353553391,0.612372436,0.612372436,-0.353553391],[-1,-1,0,0],[9E+09,9E+09,9E+09,9E+09,9E+09,9E+09]];
    CONST robtarget Target_1840:=[[124.955,124.236,0],[0.353553391,0.612372436,0.612372436,-0.353553391],[-1,-1,0,0],[9E+09,9E+09,9E+09,9E+09,9E+09,9E+09]];
    CONST robtarget Target_1850:=[[124.996,122.121,0],[0.353553391,0.612372436,0.612372436,-0.353553391],[-1,-1,0,0],[9E+09,9E+09,9E+09,9E+09,9E+09,9E+09]];
    CONST robtarget Target_1860:=[[124.996,120.424,0],[0.353553391,0.612372436,0.612372436,-0.353553391],[-1,-1,0,0],[9E+09,9E+09,9E+09,9E+09,9E+09,9E+09]];
    CONST robtarget Target_1870:=[[124.996,120.424,10],[0.353553391,0.612372436,0.612372436,-0.353553391],[-1,-1,0,0],[9E+09,9E+09,9E+09,9E+09,9E+09,9E+09]];
    CONST robtarget Target_1880:=[[48.093,102.54,10],[0.353553391,0.612372436,0.612372436,-0.353553391],[-2,0,-1,0],[9E+09,9E+09,9E+09,9E+09,9E+09,9E+09]];
    CONST robtarget Target_1890:=[[48.093,102.54,0],[0.353553391,0.612372436,0.612372436,-0.353553391],[-2,0,-1,0],[9E+09,9E+09,9E+09,9E+09,9E+09,9E+09]];
    CONST robtarget Target_1900:=[[43.231,104.473,0],[0.353553391,0.612372436,0.612372436,-0.353553391],[-2,0,-1,0],[9E+09,9E+09,9E+09,9E+09,9E+09,9E+09]];
    CONST robtarget Target_1910:=[[37.105,105.19,0],[0.353553391,0.612372436,0.612372436,-0.353553391],[-2,0,-1,0],[9E+09,9E+09,9E+09,9E+09,9E+09,9E+09]];
    CONST robtarget Target_1920:=[[32.913,104.788,0],[0.353553391,0.612372436,0.612372436,-0.353553391],[-2,0,-1,0],[9E+09,9E+09,9E+09,9E+09,9E+09,9E+09]];
    CONST robtarget Target_1930:=[[30.425,104.066,0],[0.353553391,0.612372436,0.612372436,-0.353553391],[-2,0,-1,0],[9E+09,9E+09,9E+09,9E+09,9E+09,9E+09]];
    CONST robtarget Target_1940:=[[27.453,102.491,0],[0.353553391,0.612372436,0.612372436,-0.353553391],[-2,0,-1,0],[9E+09,9E+09,9E+09,9E+09,9E+09,9E+09]];
    CONST robtarget Target_1950:=[[25.682,101,0],[0.353553391,0.612372436,0.612372436,-0.353553391],[-2,0,-1,0],[9E+09,9E+09,9E+09,9E+09,9E+09,9E+09]];
    CONST robtarget Target_1960:=[[24.18,99.225,0],[0.353553391,0.612372436,0.612372436,-0.353553391],[-2,0,-1,0],[9E+09,9E+09,9E+09,9E+09,9E+09,9E+09]];
    CONST robtarget Target_1970:=[[23.043,97.314,0],[0.353553391,0.612372436,0.612372436,-0.353553391],[-2,0,-1,0],[9E+09,9E+09,9E+09,9E+09,9E+09,9E+09]];
    CONST robtarget Target_1980:=[[22.382,95.73,0],[0.353553391,0.612372436,0.612372436,-0.353553391],[-2,0,-1,0],[9E+09,9E+09,9E+09,9E+09,9E+09,9E+09]];
    CONST robtarget Target_1990:=[[21.885,93.998,0],[0.353553391,0.612372436,0.612372436,-0.353553391],[-2,0,-1,0],[9E+09,9E+09,9E+09,9E+09,9E+09,9E+09]];
    CONST robtarget Target_2000:=[[21.534,91.845,0],[0.353553391,0.612372436,0.612372436,-0.353553391],[-2,0,-1,0],[9E+09,9E+09,9E+09,9E+09,9E+09,9E+09]];
    CONST robtarget Target_2010:=[[21.424,89.631,0],[0.353553391,0.612372436,0.612372436,-0.353553391],[-2,0,-1,0],[9E+09,9E+09,9E+09,9E+09,9E+09,9E+09]];
    CONST robtarget Target_2020:=[[21.598,86.718,0],[0.353553391,0.612372436,0.612372436,-0.353553391],[-2,0,-1,0],[9E+09,9E+09,9E+09,9E+09,9E+09,9E+09]];
    CONST robtarget Target_2030:=[[22.061,84.31,0],[0.353553391,0.612372436,0.612372436,-0.353553391],[-2,0,-1,0],[9E+09,9E+09,9E+09,9E+09,9E+09,9E+09]];
    CONST robtarget Target_2040:=[[22.438,83.089,0],[0.353553391,0.612372436,0.612372436,-0.353553391],[-2,0,-1,0],[9E+09,9E+09,9E+09,9E+09,9E+09,9E+09]];
    CONST robtarget Target_2050:=[[23.52,80.745,0],[0.353553391,0.612372436,0.612372436,-0.353553391],[-2,0,-1,0],[9E+09,9E+09,9E+09,9E+09,9E+09,9E+09]];
    CONST robtarget Target_2060:=[[25.622,78.054,0],[0.353553391,0.612372436,0.612372436,-0.353553391],[-2,0,-1,0],[9E+09,9E+09,9E+09,9E+09,9E+09,9E+09]];
    CONST robtarget Target_2070:=[[28.684,75.816,0],[0.353553391,0.612372436,0.612372436,-0.353553391],[-2,0,-1,0],[9E+09,9E+09,9E+09,9E+09,9E+09,9E+09]];
    CONST robtarget Target_2080:=[[31.534,74.671,0],[0.353553391,0.612372436,0.612372436,-0.353553391],[-2,0,-1,0],[9E+09,9E+09,9E+09,9E+09,9E+09,9E+09]];
    CONST robtarget Target_2090:=[[35.573,74.011,0],[0.353553391,0.612372436,0.612372436,-0.353553391],[-2,0,-1,0],[9E+09,9E+09,9E+09,9E+09,9E+09,9E+09]];
    CONST robtarget Target_2100:=[[38.167,74.008,0],[0.353553391,0.612372436,0.612372436,-0.353553391],[-2,0,-1,0],[9E+09,9E+09,9E+09,9E+09,9E+09,9E+09]];
    CONST robtarget Target_2110:=[[40.483,74.234,0],[0.353553391,0.612372436,0.612372436,-0.353553391],[-2,0,-1,0],[9E+09,9E+09,9E+09,9E+09,9E+09,9E+09]];
    CONST robtarget Target_2120:=[[43.194,74.764,0],[0.353553391,0.612372436,0.612372436,-0.353553391],[-2,0,-1,0],[9E+09,9E+09,9E+09,9E+09,9E+09,9E+09]];
    CONST robtarget Target_2130:=[[46.412,75.66,0],[0.353553391,0.612372436,0.612372436,-0.353553391],[-2,0,-1,0],[9E+09,9E+09,9E+09,9E+09,9E+09,9E+09]];
    CONST robtarget Target_2140:=[[48.215,76.308,0],[0.353553391,0.612372436,0.612372436,-0.353553391],[-2,0,-1,0],[9E+09,9E+09,9E+09,9E+09,9E+09,9E+09]];
    CONST robtarget Target_2150:=[[48.215,91.09,0],[0.353553391,0.612372436,0.612372436,-0.353553391],[-2,0,-1,0],[9E+09,9E+09,9E+09,9E+09,9E+09,9E+09]];
    CONST robtarget Target_2160:=[[35.111,91.09,0],[0.353553391,0.612372436,0.612372436,-0.353553391],[-2,0,-1,0],[9E+09,9E+09,9E+09,9E+09,9E+09,9E+09]];
    CONST robtarget Target_2170:=[[35.111,85.474,0],[0.353553391,0.612372436,0.612372436,-0.353553391],[-2,0,-1,0],[9E+09,9E+09,9E+09,9E+09,9E+09,9E+09]];
    CONST robtarget Target_2180:=[[40.922,85.474,0],[0.353553391,0.612372436,0.612372436,-0.353553391],[-2,0,-1,0],[9E+09,9E+09,9E+09,9E+09,9E+09,9E+09]];
    CONST robtarget Target_2190:=[[40.922,79.566,0],[0.353553391,0.612372436,0.612372436,-0.353553391],[-2,0,-1,0],[9E+09,9E+09,9E+09,9E+09,9E+09,9E+09]];
    CONST robtarget Target_2200:=[[39.025,79.493,0],[0.353553391,0.612372436,0.612372436,-0.353553391],[-2,0,-1,0],[9E+09,9E+09,9E+09,9E+09,9E+09,9E+09]];
    CONST robtarget Target_2210:=[[35.542,79.935,0],[0.353553391,0.612372436,0.612372436,-0.353553391],[-2,0,-1,0],[9E+09,9E+09,9E+09,9E+09,9E+09,9E+09]];
    CONST robtarget Target_2220:=[[32.97,81.097,0],[0.353553391,0.612372436,0.612372436,-0.353553391],[-2,0,-1,0],[9E+09,9E+09,9E+09,9E+09,9E+09,9E+09]];
    CONST robtarget Target_2230:=[[30.756,83.312,0],[0.353553391,0.612372436,0.612372436,-0.353553391],[-2,0,-1,0],[9E+09,9E+09,9E+09,9E+09,9E+09,9E+09]];
    CONST robtarget Target_2240:=[[29.841,85.252,0],[0.353553391,0.612372436,0.612372436,-0.353553391],[-2,0,-1,0],[9E+09,9E+09,9E+09,9E+09,9E+09,9E+09]];
    CONST robtarget Target_2250:=[[29.28,88.046,0],[0.353553391,0.612372436,0.612372436,-0.353553391],[-2,0,-1,0],[9E+09,9E+09,9E+09,9E+09,9E+09,9E+09]];
    CONST robtarget Target_2260:=[[29.205,89.501,0],[0.353553391,0.612372436,0.612372436,-0.353553391],[-2,0,-1,0],[9E+09,9E+09,9E+09,9E+09,9E+09,9E+09]];
    CONST robtarget Target_2270:=[[29.324,91.697,0],[0.353553391,0.612372436,0.612372436,-0.353553391],[-2,0,-1,0],[9E+09,9E+09,9E+09,9E+09,9E+09,9E+09]];
    CONST robtarget Target_2280:=[[30.172,94.739,0],[0.353553391,0.612372436,0.612372436,-0.353553391],[-2,0,-1,0],[9E+09,9E+09,9E+09,9E+09,9E+09,9E+09]];
    CONST robtarget Target_2290:=[[31.657,97.014,0],[0.353553391,0.612372436,0.612372436,-0.353553391],[-2,0,-1,0],[9E+09,9E+09,9E+09,9E+09,9E+09,9E+09]];
    CONST robtarget Target_2300:=[[33.883,98.67,0],[0.353553391,0.612372436,0.612372436,-0.353553391],[-2,0,-1,0],[9E+09,9E+09,9E+09,9E+09,9E+09,9E+09]];
    CONST robtarget Target_2310:=[[35.769,99.342,0],[0.353553391,0.612372436,0.612372436,-0.353553391],[-2,0,-1,0],[9E+09,9E+09,9E+09,9E+09,9E+09,9E+09]];
    CONST robtarget Target_2320:=[[37.808,99.594,0],[0.353553391,0.612372436,0.612372436,-0.353553391],[-2,0,-1,0],[9E+09,9E+09,9E+09,9E+09,9E+09,9E+09]];
    CONST robtarget Target_2330:=[[40.664,99.302,0],[0.353553391,0.612372436,0.612372436,-0.353553391],[-2,0,-1,0],[9E+09,9E+09,9E+09,9E+09,9E+09,9E+09]];
    CONST robtarget Target_2340:=[[43.731,98.095,0],[0.353553391,0.612372436,0.612372436,-0.353553391],[-2,0,-1,0],[9E+09,9E+09,9E+09,9E+09,9E+09,9E+09]];
    CONST robtarget Target_2350:=[[47.413,95.49,0],[0.353553391,0.612372436,0.612372436,-0.353553391],[-2,0,-1,0],[9E+09,9E+09,9E+09,9E+09,9E+09,9E+09]];
    CONST robtarget Target_2360:=[[48.093,95.49,0],[0.353553391,0.612372436,0.612372436,-0.353553391],[-2,0,-1,0],[9E+09,9E+09,9E+09,9E+09,9E+09,9E+09]];
    CONST robtarget Target_2370:=[[48.093,102.54,0],[0.353553391,0.612372436,0.612372436,-0.353553391],[-2,0,-1,0],[9E+09,9E+09,9E+09,9E+09,9E+09,9E+09]];
    CONST robtarget Target_2380:=[[48.093,102.54,10],[0.353553391,0.612372436,0.612372436,-0.353553391],[-2,0,-1,0],[9E+09,9E+09,9E+09,9E+09,9E+09,9E+09]];
    CONST robtarget Target_2390:=[[53.685,96.754,10],[0.353553391,0.612372436,0.612372436,-0.353553391],[-2,0,-1,0],[9E+09,9E+09,9E+09,9E+09,9E+09,9E+09]];
    CONST robtarget Target_2400:=[[53.685,96.754,0],[0.353553391,0.612372436,0.612372436,-0.353553391],[-2,0,-1,0],[9E+09,9E+09,9E+09,9E+09,9E+09,9E+09]];
    CONST robtarget Target_2410:=[[61.781,97.872,0],[0.353553391,0.612372436,0.612372436,-0.353553391],[-2,0,-1,0],[9E+09,9E+09,9E+09,9E+09,9E+09,9E+09]];
    CONST robtarget Target_2420:=[[66.233,97.509,0],[0.353553391,0.612372436,0.612372436,-0.353553391],[-2,0,-1,0],[9E+09,9E+09,9E+09,9E+09,9E+09,9E+09]];
    CONST robtarget Target_2430:=[[70.243,95.961,0],[0.353553391,0.612372436,0.612372436,-0.353553391],[-2,0,-1,0],[9E+09,9E+09,9E+09,9E+09,9E+09,9E+09]];
    CONST robtarget Target_2440:=[[72.614,92.613,0],[0.353553391,0.612372436,0.612372436,-0.353553391],[-2,0,-1,0],[9E+09,9E+09,9E+09,9E+09,9E+09,9E+09]];
    CONST robtarget Target_2450:=[[72.964,89.996,0],[0.353553391,0.612372436,0.612372436,-0.353553391],[-2,0,-1,0],[9E+09,9E+09,9E+09,9E+09,9E+09,9E+09]];
    CONST robtarget Target_2460:=[[72.964,74.607,0],[0.353553391,0.612372436,0.612372436,-0.353553391],[-2,0,-1,0],[9E+09,9E+09,9E+09,9E+09,9E+09,9E+09]];
    CONST robtarget Target_2470:=[[65.962,74.607,0],[0.353553391,0.612372436,0.612372436,-0.353553391],[-2,0,-1,0],[9E+09,9E+09,9E+09,9E+09,9E+09,9E+09]];
    CONST robtarget Target_2480:=[[65.962,77.013,0],[0.353553391,0.612372436,0.612372436,-0.353553391],[-2,0,-1,0],[9E+09,9E+09,9E+09,9E+09,9E+09,9E+09]];
    CONST robtarget Target_2490:=[[63.118,74.947,0],[0.353553391,0.612372436,0.612372436,-0.353553391],[-2,0,-1,0],[9E+09,9E+09,9E+09,9E+09,9E+09,9E+09]];
    CONST robtarget Target_2500:=[[58.766,73.999,0],[0.353553391,0.612372436,0.612372436,-0.353553391],[-2,0,-1,0],[9E+09,9E+09,9E+09,9E+09,9E+09,9E+09]];
    CONST robtarget Target_2510:=[[55.832,74.578,0],[0.353553391,0.612372436,0.612372436,-0.353553391],[-2,0,-1,0],[9E+09,9E+09,9E+09,9E+09,9E+09,9E+09]];
    CONST robtarget Target_2520:=[[53.483,76.327,0],[0.353553391,0.612372436,0.612372436,-0.353553391],[-2,0,-1,0],[9E+09,9E+09,9E+09,9E+09,9E+09,9E+09]];
    CONST robtarget Target_2530:=[[52.081,78.898,0],[0.353553391,0.612372436,0.612372436,-0.353553391],[-2,0,-1,0],[9E+09,9E+09,9E+09,9E+09,9E+09,9E+09]];
    CONST robtarget Target_2540:=[[51.789,81.098,0],[0.353553391,0.612372436,0.612372436,-0.353553391],[-2,0,-1,0],[9E+09,9E+09,9E+09,9E+09,9E+09,9E+09]];
    CONST robtarget Target_2550:=[[51.983,83.114,0],[0.353553391,0.612372436,0.612372436,-0.353553391],[-2,0,-1,0],[9E+09,9E+09,9E+09,9E+09,9E+09,9E+09]];
    CONST robtarget Target_2560:=[[52.864,85.258,0],[0.353553391,0.612372436,0.612372436,-0.353553391],[-2,0,-1,0],[9E+09,9E+09,9E+09,9E+09,9E+09,9E+09]];
    CONST robtarget Target_2570:=[[54.039,86.559,0],[0.353553391,0.612372436,0.612372436,-0.353553391],[-2,0,-1,0],[9E+09,9E+09,9E+09,9E+09,9E+09,9E+09]];
    CONST robtarget Target_2580:=[[55.703,87.613,0],[0.353553391,0.612372436,0.612372436,-0.353553391],[-2,0,-1,0],[9E+09,9E+09,9E+09,9E+09,9E+09,9E+09]];
    CONST robtarget Target_2590:=[[58.542,88.585,0],[0.353553391,0.612372436,0.612372436,-0.353553391],[-2,0,-1,0],[9E+09,9E+09,9E+09,9E+09,9E+09,9E+09]];
    CONST robtarget Target_2600:=[[60.612,88.946,0],[0.353553391,0.612372436,0.612372436,-0.353553391],[-2,0,-1,0],[9E+09,9E+09,9E+09,9E+09,9E+09,9E+09]];
    CONST robtarget Target_2610:=[[64.587,89.359,0],[0.353553391,0.612372436,0.612372436,-0.353553391],[-2,0,-1,0],[9E+09,9E+09,9E+09,9E+09,9E+09,9E+09]];
    CONST robtarget Target_2620:=[[66.011,89.461,0],[0.353553391,0.612372436,0.612372436,-0.353553391],[-2,0,-1,0],[9E+09,9E+09,9E+09,9E+09,9E+09,9E+09]];
    CONST robtarget Target_2630:=[[66.011,89.582,0],[0.353553391,0.612372436,0.612372436,-0.353553391],[-2,0,-1,0],[9E+09,9E+09,9E+09,9E+09,9E+09,9E+09]];
    CONST robtarget Target_2640:=[[64.625,92.171,0],[0.353553391,0.612372436,0.612372436,-0.353553391],[-2,0,-1,0],[9E+09,9E+09,9E+09,9E+09,9E+09,9E+09]];
    CONST robtarget Target_2650:=[[60.468,92.889,0],[0.353553391,0.612372436,0.612372436,-0.353553391],[-2,0,-1,0],[9E+09,9E+09,9E+09,9E+09,9E+09,9E+09]];
    CONST robtarget Target_2660:=[[54.293,91.284,0],[0.353553391,0.612372436,0.612372436,-0.353553391],[-2,0,-1,0],[9E+09,9E+09,9E+09,9E+09,9E+09,9E+09]];
    CONST robtarget Target_2670:=[[53.685,91.284,0],[0.353553391,0.612372436,0.612372436,-0.353553391],[-2,0,-1,0],[9E+09,9E+09,9E+09,9E+09,9E+09,9E+09]];
    CONST robtarget Target_2680:=[[53.685,96.754,0],[0.353553391,0.612372436,0.612372436,-0.353553391],[-2,0,-1,0],[9E+09,9E+09,9E+09,9E+09,9E+09,9E+09]];
    CONST robtarget Target_2690:=[[53.685,96.754,10],[0.353553391,0.612372436,0.612372436,-0.353553391],[-2,0,-1,0],[9E+09,9E+09,9E+09,9E+09,9E+09,9E+09]];
    CONST robtarget Target_2700:=[[65.962,85.206,10],[0.353553391,0.612372436,0.612372436,-0.353553391],[-2,0,-1,0],[9E+09,9E+09,9E+09,9E+09,9E+09,9E+09]];
    CONST robtarget Target_2710:=[[65.962,85.206,0],[0.353553391,0.612372436,0.612372436,-0.353553391],[-2,0,-1,0],[9E+09,9E+09,9E+09,9E+09,9E+09,9E+09]];
    CONST robtarget Target_2720:=[[60.881,84.38,0],[0.353553391,0.612372436,0.612372436,-0.353553391],[-2,0,-1,0],[9E+09,9E+09,9E+09,9E+09,9E+09,9E+09]];
    CONST robtarget Target_2730:=[[59.422,83.407,0],[0.353553391,0.612372436,0.612372436,-0.353553391],[-2,0,-1,0],[9E+09,9E+09,9E+09,9E+09,9E+09,9E+09]];
    CONST robtarget Target_2740:=[[58.912,81.681,0],[0.353553391,0.612372436,0.612372436,-0.353553391],[-2,0,-1,0],[9E+09,9E+09,9E+09,9E+09,9E+09,9E+09]];
    CONST robtarget Target_2750:=[[59.032,80.639,0],[0.353553391,0.612372436,0.612372436,-0.353553391],[-2,0,-1,0],[9E+09,9E+09,9E+09,9E+09,9E+09,9E+09]];
    CONST robtarget Target_2760:=[[60.054,79.339,0],[0.353553391,0.612372436,0.612372436,-0.353553391],[-2,0,-1,0],[9E+09,9E+09,9E+09,9E+09,9E+09,9E+09]];
    CONST robtarget Target_2770:=[[61.465,78.954,0],[0.353553391,0.612372436,0.612372436,-0.353553391],[-2,0,-1,0],[9E+09,9E+09,9E+09,9E+09,9E+09,9E+09]];
    CONST robtarget Target_2780:=[[62.315,78.91,0],[0.353553391,0.612372436,0.612372436,-0.353553391],[-2,0,-1,0],[9E+09,9E+09,9E+09,9E+09,9E+09,9E+09]];
    CONST robtarget Target_2790:=[[64.212,79.335,0],[0.353553391,0.612372436,0.612372436,-0.353553391],[-2,0,-1,0],[9E+09,9E+09,9E+09,9E+09,9E+09,9E+09]];
    CONST robtarget Target_2800:=[[65.962,80.514,0],[0.353553391,0.612372436,0.612372436,-0.353553391],[-2,0,-1,0],[9E+09,9E+09,9E+09,9E+09,9E+09,9E+09]];
    CONST robtarget Target_2810:=[[65.962,85.206,0],[0.353553391,0.612372436,0.612372436,-0.353553391],[-2,0,-1,0],[9E+09,9E+09,9E+09,9E+09,9E+09,9E+09]];
    CONST robtarget Target_2820:=[[65.962,85.206,10],[0.353553391,0.612372436,0.612372436,-0.353553391],[-2,0,-1,0],[9E+09,9E+09,9E+09,9E+09,9E+09,9E+09]];
    CONST robtarget Target_2830:=[[78.191,105.944,10],[0.353553391,0.612372436,0.612372436,-0.353553391],[-2,0,-1,0],[9E+09,9E+09,9E+09,9E+09,9E+09,9E+09]];
    CONST robtarget Target_2840:=[[78.191,105.944,0],[0.353553391,0.612372436,0.612372436,-0.353553391],[-2,0,-1,0],[9E+09,9E+09,9E+09,9E+09,9E+09,9E+09]];
    CONST robtarget Target_2850:=[[78.191,74.607,0],[0.353553391,0.612372436,0.612372436,-0.353553391],[-2,0,-1,0],[9E+09,9E+09,9E+09,9E+09,9E+09,9E+09]];
    CONST robtarget Target_2860:=[[84.949,74.607,0],[0.353553391,0.612372436,0.612372436,-0.353553391],[-1,0,-1,0],[9E+09,9E+09,9E+09,9E+09,9E+09,9E+09]];
    CONST robtarget Target_2870:=[[85.241,75.725,0],[0.353553391,0.612372436,0.612372436,-0.353553391],[-1,0,-1,0],[9E+09,9E+09,9E+09,9E+09,9E+09,9E+09]];
    CONST robtarget Target_2880:=[[90.832,74.169,0],[0.353553391,0.612372436,0.612372436,-0.353553391],[-1,0,-1,0],[9E+09,9E+09,9E+09,9E+09,9E+09,9E+09]];
    CONST robtarget Target_2890:=[[94.512,74.978,0],[0.353553391,0.612372436,0.612372436,-0.353553391],[-1,0,-1,0],[9E+09,9E+09,9E+09,9E+09,9E+09,9E+09]];
    CONST robtarget Target_2900:=[[97.536,77.39,0],[0.353553391,0.612372436,0.612372436,-0.353553391],[-1,-1,0,0],[9E+09,9E+09,9E+09,9E+09,9E+09,9E+09]];
    CONST robtarget Target_2910:=[[99.251,80.187,0],[0.353553391,0.612372436,0.612372436,-0.353553391],[-1,-1,0,0],[9E+09,9E+09,9E+09,9E+09,9E+09,9E+09]];
    CONST robtarget Target_2920:=[[100.173,83.531,0],[0.353553391,0.612372436,0.612372436,-0.353553391],[-1,-1,0,0],[9E+09,9E+09,9E+09,9E+09,9E+09,9E+09]];
    CONST robtarget Target_2930:=[[100.362,86.227,0],[0.353553391,0.612372436,0.612372436,-0.353553391],[-1,-1,0,0],[9E+09,9E+09,9E+09,9E+09,9E+09,9E+09]];
    CONST robtarget Target_2940:=[[100.162,89.348,0],[0.353553391,0.612372436,0.612372436,-0.353553391],[-1,-1,0,0],[9E+09,9E+09,9E+09,9E+09,9E+09,9E+09]];
    CONST robtarget Target_2950:=[[99.451,92.348,0],[0.353553391,0.612372436,0.612372436,-0.353553391],[-1,-1,0,0],[9E+09,9E+09,9E+09,9E+09,9E+09,9E+09]];
    CONST robtarget Target_2960:=[[98.126,94.909,0],[0.353553391,0.612372436,0.612372436,-0.353553391],[-1,-1,0,0],[9E+09,9E+09,9E+09,9E+09,9E+09,9E+09]];
    CONST robtarget Target_2970:=[[96.145,96.789,0],[0.353553391,0.612372436,0.612372436,-0.353553391],[-1,0,-1,0],[9E+09,9E+09,9E+09,9E+09,9E+09,9E+09]];
    CONST robtarget Target_2980:=[[93.246,97.782,0],[0.353553391,0.612372436,0.612372436,-0.353553391],[-1,0,-1,0],[9E+09,9E+09,9E+09,9E+09,9E+09,9E+09]];
    CONST robtarget Target_2990:=[[91.056,97.792,0],[0.353553391,0.612372436,0.612372436,-0.353553391],[-1,0,-1,0],[9E+09,9E+09,9E+09,9E+09,9E+09,9E+09]];
    CONST robtarget Target_3000:=[[88.708,97.17,0],[0.353553391,0.612372436,0.612372436,-0.353553391],[-1,0,-1,0],[9E+09,9E+09,9E+09,9E+09,9E+09,9E+09]];
    CONST robtarget Target_3010:=[[86.849,96.094,0],[0.353553391,0.612372436,0.612372436,-0.353553391],[-1,0,-1,0],[9E+09,9E+09,9E+09,9E+09,9E+09,9E+09]];
    CONST robtarget Target_3020:=[[85.241,94.858,0],[0.353553391,0.612372436,0.612372436,-0.353553391],[-1,0,-1,0],[9E+09,9E+09,9E+09,9E+09,9E+09,9E+09]];
    CONST robtarget Target_3030:=[[85.241,105.944,0],[0.353553391,0.612372436,0.612372436,-0.353553391],[-1,0,-1,0],[9E+09,9E+09,9E+09,9E+09,9E+09,9E+09]];
    CONST robtarget Target_3040:=[[78.191,105.944,0],[0.353553391,0.612372436,0.612372436,-0.353553391],[-2,0,-1,0],[9E+09,9E+09,9E+09,9E+09,9E+09,9E+09]];
    CONST robtarget Target_3050:=[[78.191,105.944,10],[0.353553391,0.612372436,0.612372436,-0.353553391],[-2,0,-1,0],[9E+09,9E+09,9E+09,9E+09,9E+09,9E+09]];
    CONST robtarget Target_3060:=[[85.241,91.138,10],[0.353553391,0.612372436,0.612372436,-0.353553391],[-1,0,-1,0],[9E+09,9E+09,9E+09,9E+09,9E+09,9E+09]];
    CONST robtarget Target_3070:=[[85.241,91.138,0],[0.353553391,0.612372436,0.612372436,-0.353553391],[-1,0,-1,0],[9E+09,9E+09,9E+09,9E+09,9E+09,9E+09]];
    CONST robtarget Target_3080:=[[85.241,79.809,0],[0.353553391,0.612372436,0.612372436,-0.353553391],[-1,0,-1,0],[9E+09,9E+09,9E+09,9E+09,9E+09,9E+09]];
    CONST robtarget Target_3090:=[[88.085,79.323,0],[0.353553391,0.612372436,0.612372436,-0.353553391],[-1,0,-1,0],[9E+09,9E+09,9E+09,9E+09,9E+09,9E+09]];
    CONST robtarget Target_3100:=[[90.106,79.66,0],[0.353553391,0.612372436,0.612372436,-0.353553391],[-1,0,-1,0],[9E+09,9E+09,9E+09,9E+09,9E+09,9E+09]];
    CONST robtarget Target_3110:=[[91.905,81.033,0],[0.353553391,0.612372436,0.612372436,-0.353553391],[-1,0,-1,0],[9E+09,9E+09,9E+09,9E+09,9E+09,9E+09]];
    CONST robtarget Target_3120:=[[92.891,83.394,0],[0.353553391,0.612372436,0.612372436,-0.353553391],[-1,0,-1,0],[9E+09,9E+09,9E+09,9E+09,9E+09,9E+09]];
    CONST robtarget Target_3130:=[[93.142,86.082,0],[0.353553391,0.612372436,0.612372436,-0.353553391],[-1,0,-1,0],[9E+09,9E+09,9E+09,9E+09,9E+09,9E+09]];
    CONST robtarget Target_3140:=[[92.957,88.611,0],[0.353553391,0.612372436,0.612372436,-0.353553391],[-1,0,-1,0],[9E+09,9E+09,9E+09,9E+09,9E+09,9E+09]];
    CONST robtarget Target_3150:=[[92.311,90.605,0],[0.353553391,0.612372436,0.612372436,-0.353553391],[-1,0,-1,0],[9E+09,9E+09,9E+09,9E+09,9E+09,9E+09]];
    CONST robtarget Target_3160:=[[90.724,92.035,0],[0.353553391,0.612372436,0.612372436,-0.353553391],[-1,0,-1,0],[9E+09,9E+09,9E+09,9E+09,9E+09,9E+09]];
    CONST robtarget Target_3170:=[[88.961,92.354,0],[0.353553391,0.612372436,0.612372436,-0.353553391],[-1,0,-1,0],[9E+09,9E+09,9E+09,9E+09,9E+09,9E+09]];
    CONST robtarget Target_3180:=[[87.176,92.081,0],[0.353553391,0.612372436,0.612372436,-0.353553391],[-1,0,-1,0],[9E+09,9E+09,9E+09,9E+09,9E+09,9E+09]];
    CONST robtarget Target_3190:=[[85.241,91.138,0],[0.353553391,0.612372436,0.612372436,-0.353553391],[-1,0,-1,0],[9E+09,9E+09,9E+09,9E+09,9E+09,9E+09]];
    CONST robtarget Target_3200:=[[85.241,91.138,10],[0.353553391,0.612372436,0.612372436,-0.353553391],[-1,0,-1,0],[9E+09,9E+09,9E+09,9E+09,9E+09,9E+09]];
    CONST robtarget Target_3210:=[[114.293,92.889,10],[0.353553391,0.612372436,0.612372436,-0.353553391],[-1,-1,0,0],[9E+09,9E+09,9E+09,9E+09,9E+09,9E+09]];
    CONST robtarget Target_3220:=[[114.293,92.889,0],[0.353553391,0.612372436,0.612372436,-0.353553391],[-1,-1,0,0],[9E+09,9E+09,9E+09,9E+09,9E+09,9E+09]];
    CONST robtarget Target_3230:=[[111.516,91.894,0],[0.353553391,0.612372436,0.612372436,-0.353553391],[-1,-1,0,0],[9E+09,9E+09,9E+09,9E+09,9E+09,9E+09]];
    CONST robtarget Target_3240:=[[110.079,88.878,0],[0.353553391,0.612372436,0.612372436,-0.353553391],[-1,-1,0,0],[9E+09,9E+09,9E+09,9E+09,9E+09,9E+09]];
    CONST robtarget Target_3250:=[[109.82,85.731,0],[0.353553391,0.612372436,0.612372436,-0.353553391],[-1,-1,0,0],[9E+09,9E+09,9E+09,9E+09,9E+09,9E+09]];
    CONST robtarget Target_3260:=[[110.134,82.622,0],[0.353553391,0.612372436,0.612372436,-0.353553391],[-1,-1,0,0],[9E+09,9E+09,9E+09,9E+09,9E+09,9E+09]];
    CONST robtarget Target_3270:=[[112.748,79.215,0],[0.353553391,0.612372436,0.612372436,-0.353553391],[-1,-1,0,0],[9E+09,9E+09,9E+09,9E+09,9E+09,9E+09]];
    CONST robtarget Target_3280:=[[115.472,79.116,0],[0.353553391,0.612372436,0.612372436,-0.353553391],[-1,-1,0,0],[9E+09,9E+09,9E+09,9E+09,9E+09,9E+09]];
    CONST robtarget Target_3290:=[[117.853,81.029,0],[0.353553391,0.612372436,0.612372436,-0.353553391],[-1,-1,0,0],[9E+09,9E+09,9E+09,9E+09,9E+09,9E+09]];
    CONST robtarget Target_3300:=[[118.692,84.329,0],[0.353553391,0.612372436,0.612372436,-0.353553391],[-1,-1,0,0],[9E+09,9E+09,9E+09,9E+09,9E+09,9E+09]];
    CONST robtarget Target_3310:=[[118.705,87.144,0],[0.353553391,0.612372436,0.612372436,-0.353553391],[-1,-1,0,0],[9E+09,9E+09,9E+09,9E+09,9E+09,9E+09]];
    CONST robtarget Target_3320:=[[117.699,91.082,0],[0.353553391,0.612372436,0.612372436,-0.353553391],[-1,-1,0,0],[9E+09,9E+09,9E+09,9E+09,9E+09,9E+09]];
    CONST robtarget Target_3330:=[[116.9,92.042,0],[0.353553391,0.612372436,0.612372436,-0.353553391],[-1,-1,0,0],[9E+09,9E+09,9E+09,9E+09,9E+09,9E+09]];
    CONST robtarget Target_3340:=[[114.293,92.889,0],[0.353553391,0.612372436,0.612372436,-0.353553391],[-1,-1,0,0],[9E+09,9E+09,9E+09,9E+09,9E+09,9E+09]];
    CONST robtarget Target_3350:=[[114.293,92.889,10],[0.353553391,0.612372436,0.612372436,-0.353553391],[-1,-1,0,0],[9E+09,9E+09,9E+09,9E+09,9E+09,9E+09]];
    CONST robtarget Target_3360:=[[114.293,97.945,10],[0.353553391,0.612372436,0.612372436,-0.353553391],[-1,-1,0,0],[9E+09,9E+09,9E+09,9E+09,9E+09,9E+09]];
    CONST robtarget Target_3370:=[[114.293,97.945,0],[0.353553391,0.612372436,0.612372436,-0.353553391],[-1,-1,0,0],[9E+09,9E+09,9E+09,9E+09,9E+09,9E+09]];
    CONST robtarget Target_3380:=[[119.425,97.063,0],[0.353553391,0.612372436,0.612372436,-0.353553391],[-1,-1,0,0],[9E+09,9E+09,9E+09,9E+09,9E+09,9E+09]];
    CONST robtarget Target_3390:=[[122.854,94.783,0],[0.353553391,0.612372436,0.612372436,-0.353553391],[-1,-1,0,0],[9E+09,9E+09,9E+09,9E+09,9E+09,9E+09]];
    CONST robtarget Target_3400:=[[124.981,91.496,0],[0.353553391,0.612372436,0.612372436,-0.353553391],[-1,-1,0,0],[9E+09,9E+09,9E+09,9E+09,9E+09,9E+09]];
    CONST robtarget Target_3410:=[[125.918,87.222,0],[0.353553391,0.612372436,0.612372436,-0.353553391],[-1,-1,0,0],[9E+09,9E+09,9E+09,9E+09,9E+09,9E+09]];
    CONST robtarget Target_3420:=[[125.74,83.065,0],[0.353553391,0.612372436,0.612372436,-0.353553391],[-1,-1,0,0],[9E+09,9E+09,9E+09,9E+09,9E+09,9E+09]];
    CONST robtarget Target_3430:=[[124.292,78.941,0],[0.353553391,0.612372436,0.612372436,-0.353553391],[-1,-1,0,0],[9E+09,9E+09,9E+09,9E+09,9E+09,9E+09]];
    CONST robtarget Target_3440:=[[122.614,76.811,0],[0.353553391,0.612372436,0.612372436,-0.353553391],[-1,-1,0,0],[9E+09,9E+09,9E+09,9E+09,9E+09,9E+09]];
    CONST robtarget Target_3450:=[[118.869,74.576,0],[0.353553391,0.612372436,0.612372436,-0.353553391],[-1,-1,0,0],[9E+09,9E+09,9E+09,9E+09,9E+09,9E+09]];
    CONST robtarget Target_3460:=[[115.671,73.954,0],[0.353553391,0.612372436,0.612372436,-0.353553391],[-1,-1,0,0],[9E+09,9E+09,9E+09,9E+09,9E+09,9E+09]];
    CONST robtarget Target_3470:=[[111.694,74.099,0],[0.353553391,0.612372436,0.612372436,-0.353553391],[-1,-1,0,0],[9E+09,9E+09,9E+09,9E+09,9E+09,9E+09]];
    CONST robtarget Target_3480:=[[107.574,75.575,0],[0.353553391,0.612372436,0.612372436,-0.353553391],[-1,-1,0,0],[9E+09,9E+09,9E+09,9E+09,9E+09,9E+09]];
    CONST robtarget Target_3490:=[[104.577,78.476,0],[0.353553391,0.612372436,0.612372436,-0.353553391],[-1,-1,0,0],[9E+09,9E+09,9E+09,9E+09,9E+09,9E+09]];
    CONST robtarget Target_3500:=[[103.102,81.78,0],[0.353553391,0.612372436,0.612372436,-0.353553391],[-1,-1,0,0],[9E+09,9E+09,9E+09,9E+09,9E+09,9E+09]];
    CONST robtarget Target_3510:=[[102.673,84.234,0],[0.353553391,0.612372436,0.612372436,-0.353553391],[-1,-1,0,0],[9E+09,9E+09,9E+09,9E+09,9E+09,9E+09]];
    CONST robtarget Target_3520:=[[102.712,87.979,0],[0.353553391,0.612372436,0.612372436,-0.353553391],[-1,-1,0,0],[9E+09,9E+09,9E+09,9E+09,9E+09,9E+09]];
    CONST robtarget Target_3530:=[[103.395,91.017,0],[0.353553391,0.612372436,0.612372436,-0.353553391],[-1,-1,0,0],[9E+09,9E+09,9E+09,9E+09,9E+09,9E+09]];
    CONST robtarget Target_3540:=[[104.511,93.286,0],[0.353553391,0.612372436,0.612372436,-0.353553391],[-1,-1,0,0],[9E+09,9E+09,9E+09,9E+09,9E+09,9E+09]];
    CONST robtarget Target_3550:=[[106.651,95.634,0],[0.353553391,0.612372436,0.612372436,-0.353553391],[-1,-1,0,0],[9E+09,9E+09,9E+09,9E+09,9E+09,9E+09]];
    CONST robtarget Target_3560:=[[109.412,97.163,0],[0.353553391,0.612372436,0.612372436,-0.353553391],[-1,-1,0,0],[9E+09,9E+09,9E+09,9E+09,9E+09,9E+09]];
    CONST robtarget Target_3570:=[[114.293,97.945,0],[0.353553391,0.612372436,0.612372436,-0.353553391],[-1,-1,0,0],[9E+09,9E+09,9E+09,9E+09,9E+09,9E+09]];
    CONST robtarget Target_3580:=[[114.293,97.945,10],[0.353553391,0.612372436,0.612372436,-0.353553391],[-1,-1,0,0],[9E+09,9E+09,9E+09,9E+09,9E+09,9E+09]];
    CONST robtarget Target_3590:=[[57.132,66.1,10],[0.353553391,0.612372436,0.612372436,-0.353553391],[-2,0,-1,0],[9E+09,9E+09,9E+09,9E+09,9E+09,9E+09]];
    CONST robtarget Target_3600:=[[57.132,66.1,0],[0.353553391,0.612372436,0.612372436,-0.353553391],[-2,0,-1,0],[9E+09,9E+09,9E+09,9E+09,9E+09,9E+09]];
    CONST robtarget Target_3610:=[[40.852,48.713,0],[0.353553391,0.612372436,0.612372436,-0.353553391],[-2,0,-1,0],[9E+09,9E+09,9E+09,9E+09,9E+09,9E+09]];
    CONST robtarget Target_3620:=[[40.852,45.296,0],[0.353553391,0.612372436,0.612372436,-0.353553391],[-2,0,-1,0],[9E+09,9E+09,9E+09,9E+09,9E+09,9E+09]];
    CONST robtarget Target_3630:=[[75,4.113,0],[0.353553391,0.612372436,0.612372436,-0.353553391],[-2,0,-1,0],[9E+09,9E+09,9E+09,9E+09,9E+09,9E+09]];
    CONST robtarget Target_3640:=[[109.148,45.296,0],[0.353553391,0.612372436,0.612372436,-0.353553391],[-1,-1,0,0],[9E+09,9E+09,9E+09,9E+09,9E+09,9E+09]];
    CONST robtarget Target_3650:=[[109.148,48.713,0],[0.353553391,0.612372436,0.612372436,-0.353553391],[-1,-1,0,0],[9E+09,9E+09,9E+09,9E+09,9E+09,9E+09]];
    CONST robtarget Target_3660:=[[92.868,66.1,0],[0.353553391,0.612372436,0.612372436,-0.353553391],[-1,0,-1,0],[9E+09,9E+09,9E+09,9E+09,9E+09,9E+09]];
    CONST robtarget Target_3670:=[[57.132,66.1,0],[0.353553391,0.612372436,0.612372436,-0.353553391],[-2,0,-1,0],[9E+09,9E+09,9E+09,9E+09,9E+09,9E+09]];
    CONST robtarget Target_3680:=[[57.132,66.1,10],[0.353553391,0.612372436,0.612372436,-0.353553391],[-2,0,-1,0],[9E+09,9E+09,9E+09,9E+09,9E+09,9E+09]];
    CONST robtarget Target_3690:=[[59.3,61.1,10],[0.353553391,0.612372436,0.612372436,-0.353553391],[-2,0,-1,0],[9E+09,9E+09,9E+09,9E+09,9E+09,9E+09]];
    CONST robtarget Target_3700:=[[59.3,61.1,0],[0.353553391,0.612372436,0.612372436,-0.353553391],[-2,0,-1,0],[9E+09,9E+09,9E+09,9E+09,9E+09,9E+09]];
    CONST robtarget Target_3710:=[[48.446,49.508,0],[0.353553391,0.612372436,0.612372436,-0.353553391],[-2,0,-1,0],[9E+09,9E+09,9E+09,9E+09,9E+09,9E+09]];
    CONST robtarget Target_3720:=[[59.481,49.508,0],[0.353553391,0.612372436,0.612372436,-0.353553391],[-2,0,-1,0],[9E+09,9E+09,9E+09,9E+09,9E+09,9E+09]];
    CONST robtarget Target_3730:=[[69.526,61.1,0],[0.353553391,0.612372436,0.612372436,-0.353553391],[-2,0,-1,0],[9E+09,9E+09,9E+09,9E+09,9E+09,9E+09]];
    CONST robtarget Target_3740:=[[59.3,61.1,0],[0.353553391,0.612372436,0.612372436,-0.353553391],[-2,0,-1,0],[9E+09,9E+09,9E+09,9E+09,9E+09,9E+09]];
    CONST robtarget Target_3750:=[[59.3,61.1,10],[0.353553391,0.612372436,0.612372436,-0.353553391],[-2,0,-1,0],[9E+09,9E+09,9E+09,9E+09,9E+09,9E+09]];
    CONST robtarget Target_3760:=[[80.474,61.1,10],[0.353553391,0.612372436,0.612372436,-0.353553391],[-2,0,-1,0],[9E+09,9E+09,9E+09,9E+09,9E+09,9E+09]];
    CONST robtarget Target_3770:=[[80.474,61.1,0],[0.353553391,0.612372436,0.612372436,-0.353553391],[-2,0,-1,0],[9E+09,9E+09,9E+09,9E+09,9E+09,9E+09]];
    CONST robtarget Target_3780:=[[90.7,61.1,0],[0.353553391,0.612372436,0.612372436,-0.353553391],[-1,0,-1,0],[9E+09,9E+09,9E+09,9E+09,9E+09,9E+09]];
    CONST robtarget Target_3790:=[[101.554,49.508,0],[0.353553391,0.612372436,0.612372436,-0.353553391],[-1,-1,0,0],[9E+09,9E+09,9E+09,9E+09,9E+09,9E+09]];
    CONST robtarget Target_3800:=[[90.519,49.508,0],[0.353553391,0.612372436,0.612372436,-0.353553391],[-1,0,-1,0],[9E+09,9E+09,9E+09,9E+09,9E+09,9E+09]];
    CONST robtarget Target_3810:=[[80.474,61.1,0],[0.353553391,0.612372436,0.612372436,-0.353553391],[-2,0,-1,0],[9E+09,9E+09,9E+09,9E+09,9E+09,9E+09]];
    CONST robtarget Target_3820:=[[80.474,61.1,10],[0.353553391,0.612372436,0.612372436,-0.353553391],[-2,0,-1,0],[9E+09,9E+09,9E+09,9E+09,9E+09,9E+09]];
    CONST robtarget Target_3830:=[[75,59.782,10],[0.353553391,0.612372436,0.612372436,-0.353553391],[-2,0,-1,0],[9E+09,9E+09,9E+09,9E+09,9E+09,9E+09]];
    CONST robtarget Target_3840:=[[75,59.782,0],[0.353553391,0.612372436,0.612372436,-0.353553391],[-2,0,-1,0],[9E+09,9E+09,9E+09,9E+09,9E+09,9E+09]];
    CONST robtarget Target_3850:=[[83.903,49.508,0],[0.353553391,0.612372436,0.612372436,-0.353553391],[-1,0,-1,0],[9E+09,9E+09,9E+09,9E+09,9E+09,9E+09]];
    CONST robtarget Target_3860:=[[66.097,49.508,0],[0.353553391,0.612372436,0.612372436,-0.353553391],[-2,0,-1,0],[9E+09,9E+09,9E+09,9E+09,9E+09,9E+09]];
    CONST robtarget Target_3870:=[[75,59.782,0],[0.353553391,0.612372436,0.612372436,-0.353553391],[-2,0,-1,0],[9E+09,9E+09,9E+09,9E+09,9E+09,9E+09]];
    CONST robtarget Target_3880:=[[75,59.782,10],[0.353553391,0.612372436,0.612372436,-0.353553391],[-2,0,-1,0],[9E+09,9E+09,9E+09,9E+09,9E+09,9E+09]];
    CONST robtarget Target_3890:=[[64.21,44.508,10],[0.353553391,0.612372436,0.612372436,-0.353553391],[-2,0,-1,0],[9E+09,9E+09,9E+09,9E+09,9E+09,9E+09]];
    CONST robtarget Target_3900:=[[64.21,44.508,0],[0.353553391,0.612372436,0.612372436,-0.353553391],[-2,0,-1,0],[9E+09,9E+09,9E+09,9E+09,9E+09,9E+09]];
    CONST robtarget Target_3910:=[[85.79,44.508,0],[0.353553391,0.612372436,0.612372436,-0.353553391],[-1,0,-1,0],[9E+09,9E+09,9E+09,9E+09,9E+09,9E+09]];
    CONST robtarget Target_3920:=[[75,15.254,0],[0.353553391,0.612372436,0.612372436,-0.353553391],[-2,0,-1,0],[9E+09,9E+09,9E+09,9E+09,9E+09,9E+09]];
    CONST robtarget Target_3930:=[[64.21,44.508,0],[0.353553391,0.612372436,0.612372436,-0.353553391],[-2,0,-1,0],[9E+09,9E+09,9E+09,9E+09,9E+09,9E+09]];
    CONST robtarget Target_3940:=[[64.21,44.508,10],[0.353553391,0.612372436,0.612372436,-0.353553391],[-2,0,-1,0],[9E+09,9E+09,9E+09,9E+09,9E+09,9E+09]];
    CONST robtarget Target_3950:=[[58.88,44.508,10],[0.353553391,0.612372436,0.612372436,-0.353553391],[-2,0,-1,0],[9E+09,9E+09,9E+09,9E+09,9E+09,9E+09]];
    CONST robtarget Target_3960:=[[58.88,44.508,0],[0.353553391,0.612372436,0.612372436,-0.353553391],[-2,0,-1,0],[9E+09,9E+09,9E+09,9E+09,9E+09,9E+09]];
    CONST robtarget Target_3970:=[[48.001,44.508,0],[0.353553391,0.612372436,0.612372436,-0.353553391],[-2,0,-1,0],[9E+09,9E+09,9E+09,9E+09,9E+09,9E+09]];
    CONST robtarget Target_3980:=[[67.598,20.874,0],[0.353553391,0.612372436,0.612372436,-0.353553391],[-2,0,-1,0],[9E+09,9E+09,9E+09,9E+09,9E+09,9E+09]];
    CONST robtarget Target_3990:=[[58.88,44.508,0],[0.353553391,0.612372436,0.612372436,-0.353553391],[-2,0,-1,0],[9E+09,9E+09,9E+09,9E+09,9E+09,9E+09]];
    CONST robtarget Target_4000:=[[58.88,44.508,10],[0.353553391,0.612372436,0.612372436,-0.353553391],[-2,0,-1,0],[9E+09,9E+09,9E+09,9E+09,9E+09,9E+09]];
    CONST robtarget Target_4010:=[[91.12,44.508,10],[0.353553391,0.612372436,0.612372436,-0.353553391],[-1,0,-1,0],[9E+09,9E+09,9E+09,9E+09,9E+09,9E+09]];
    CONST robtarget Target_4020:=[[91.12,44.508,0],[0.353553391,0.612372436,0.612372436,-0.353553391],[-1,0,-1,0],[9E+09,9E+09,9E+09,9E+09,9E+09,9E+09]];
    CONST robtarget Target_4030:=[[101.999,44.508,0],[0.353553391,0.612372436,0.612372436,-0.353553391],[-1,-1,0,0],[9E+09,9E+09,9E+09,9E+09,9E+09,9E+09]];
    CONST robtarget Target_4040:=[[82.402,20.874,0],[0.353553391,0.612372436,0.612372436,-0.353553391],[-1,0,-1,0],[9E+09,9E+09,9E+09,9E+09,9E+09,9E+09]];
    CONST robtarget Target_4050:=[[91.12,44.508,0],[0.353553391,0.612372436,0.612372436,-0.353553391],[-1,0,-1,0],[9E+09,9E+09,9E+09,9E+09,9E+09,9E+09]];
    CONST robtarget Target_4060:=[[91.12,44.508,10],[0.353553391,0.612372436,0.612372436,-0.353553391],[-1,0,-1,0],[9E+09,9E+09,9E+09,9E+09,9E+09,9E+09]];
	!TASK PERS wobjdata cajaReal:=[FALSE,TRUE,"",[[-78.3773,-694.538,672.47],[0.999913,-0.000112558,0.000158461,0.0132015]],[[0,0,0],[1,0,0,0]]];
	TASK PERS wobjdata Caja:=[FALSE,TRUE,"",[[-78.3773,-694.538,672.47],[0.999913,-0.000112558,0.000158461,0.0132015]],[[0,0,0],[1,0,0,0]]];
    CONST robtarget Orientacion:=[[82.538787316,163.240118386,11.65819798],[0.318981086,0.637231736,0.620524538,-0.327316483],[-2,1,-1,0],[9E+09,9E+09,9E+09,9E+09,9E+09,9E+09]];
    CONST robtarget Home_cafe:=[[75,75,40],[0.353553391,0.612372436,0.612372436,-0.353553391],[-2,0,-1,0],[9E+09,9E+09,9E+09,9E+09,9E+09,9E+09]];
    CONST jointtarget Home_ABS:= [[0,0,0,0,30,0],[9E+09,9E+09,9E+09,9E+09,9E+09,9E+09]];
    CONST jointtarget Mantenimiento_Point:= [[90,0,0,0,30,0],[9E+09,9E+09,9E+09,9E+09,9E+09,9E+09]];
    TASK PERS wobjdata caja2:=[FALSE,TRUE,"",[[0,0,0],[1,0,0,0]],[[-80.4277,-562.959,675.252],[0.730832,0.00218981,0.0010399,-0.682553]]];     TASK PERS wobjdata Caja_2:=[FALSE,TRUE,"",[[-78.3773,-694.538,672.47],[0.71638,-0.000191639,3.2458E-5,-0.69771]],[[0,0,0],[1,0,0,0]]];
    CONST robtarget Target_4060_2:=[[91.12,44.508,10],[0.726314069,0.009187373,0.687236181,-0.009481395],[-1,0,-1,0],[9E+09,9E+09,9E+09,9E+09,9E+09,9E+09]];
    CONST robtarget Home_cafe_2:=[[75.000360099,74.999824312,40.000424346],[0.726314069,0.009187373,0.687236181,-0.009481395],[-2,0,-1,0],[9E+09,9E+09,9E+09,9E+09,9E+09,9E+09]];
    CONST robtarget Target_10_2:=[[0,0,0],[0.726314069,0.009187373,0.687236181,-0.009481395],[0,-1,0,0],[9E+09,9E+09,9E+09,9E+09,9E+09,9E+09]];
    CONST robtarget Target_20_2:=[[0,150,0],[0.726314069,0.009187373,0.687236181,-0.009481395],[0,-1,0,0],[9E+09,9E+09,9E+09,9E+09,9E+09,9E+09]];
    CONST robtarget Target_30_2:=[[150,150,0],[0.726314069,0.009187373,0.687236181,-0.009481395],[-1,0,-1,0],[9E+09,9E+09,9E+09,9E+09,9E+09,9E+09]];
    CONST robtarget Target_40_2:=[[150,0,0],[0.726314069,0.009187373,0.687236181,-0.009481395],[-1,0,-1,0],[9E+09,9E+09,9E+09,9E+09,9E+09,9E+09]];
    CONST robtarget Target_60_2:=[[27.192,140.457,0],[0.726314069,0.009187373,0.687236181,-0.009481395],[-2,0,-1,0],[9E+09,9E+09,9E+09,9E+09,9E+09,9E+09]];
    CONST robtarget Target_70_2:=[[35.871,140.457,0],[0.726314069,0.009187373,0.687236181,-0.009481395],[-2,0,-1,0],[9E+09,9E+09,9E+09,9E+09,9E+09,9E+09]];
    CONST robtarget Target_80_2:=[[42.532,125.651,0],[0.726314069,0.009187373,0.687236181,-0.009481395],[-2,0,-1,0],[9E+09,9E+09,9E+09,9E+09,9E+09,9E+09]];
    CONST robtarget Target_90_2:=[[49.145,140.457,0],[0.726314069,0.009187373,0.687236181,-0.009481395],[-2,0,-1,0],[9E+09,9E+09,9E+09,9E+09,9E+09,9E+09]];
    CONST robtarget Target_100_2:=[[57.824,140.457,0],[0.726314069,0.009187373,0.687236181,-0.009481395],[-2,0,-1,0],[9E+09,9E+09,9E+09,9E+09,9E+09,9E+09]];
    CONST robtarget Target_110_2:=[[57.824,110.457,0],[0.726314069,0.009187373,0.687236181,-0.009481395],[-2,0,-1,0],[9E+09,9E+09,9E+09,9E+09,9E+09,9E+09]];
    CONST robtarget Target_120_2:=[[50.336,110.457,0],[0.726314069,0.009187373,0.687236181,-0.009481395],[-2,0,-1,0],[9E+09,9E+09,9E+09,9E+09,9E+09,9E+09]];
    CONST robtarget Target_130_2:=[[50.336,130.343,0],[0.726314069,0.009187373,0.687236181,-0.009481395],[-2,0,-1,0],[9E+09,9E+09,9E+09,9E+09,9E+09,9E+09]];
    CONST robtarget Target_140_2:=[[44.891,117.507,0],[0.726314069,0.009187373,0.687236181,-0.009481395],[-2,0,-1,0],[9E+09,9E+09,9E+09,9E+09,9E+09,9E+09]];
    CONST robtarget Target_150_2:=[[39.737,117.507,0],[0.726314069,0.009187373,0.687236181,-0.009481395],[-2,0,-1,0],[9E+09,9E+09,9E+09,9E+09,9E+09,9E+09]];
    CONST robtarget Target_160_2:=[[34.291,130.343,0],[0.726314069,0.009187373,0.687236181,-0.009481395],[-2,0,-1,0],[9E+09,9E+09,9E+09,9E+09,9E+09,9E+09]];
    CONST robtarget Target_170_2:=[[34.291,110.457,0],[0.726314069,0.009187373,0.687236181,-0.009481395],[-2,0,-1,0],[9E+09,9E+09,9E+09,9E+09,9E+09,9E+09]];
    CONST robtarget Target_180_2:=[[27.192,110.457,0],[0.726314069,0.009187373,0.687236181,-0.009481395],[-2,0,-1,0],[9E+09,9E+09,9E+09,9E+09,9E+09,9E+09]];
    CONST robtarget Target_190_2:=[[27.192,140.457,0],[0.726314069,0.009187373,0.687236181,-0.009481395],[-2,0,-1,0],[9E+09,9E+09,9E+09,9E+09,9E+09,9E+09]];
    CONST robtarget Target_200_2:=[[27.192,140.457,10],[0.726314069,0.009187373,0.687236181,-0.009481395],[-2,0,-1,0],[9E+09,9E+09,9E+09,9E+09,9E+09,9E+09]];
    CONST robtarget Target_210_2:=[[63.829,132.604,10],[0.726314069,0.009187373,0.687236181,-0.009481395],[-2,0,-1,0],[9E+09,9E+09,9E+09,9E+09,9E+09,9E+09]];
    CONST robtarget Target_220_2:=[[63.829,132.604,0],[0.726314069,0.009187373,0.687236181,-0.009481395],[-2,0,-1,0],[9E+09,9E+09,9E+09,9E+09,9E+09,9E+09]];
    CONST robtarget Target_230_2:=[[71.925,133.722,0],[0.726314069,0.009187373,0.687236181,-0.009481395],[-2,0,-1,0],[9E+09,9E+09,9E+09,9E+09,9E+09,9E+09]];
    CONST robtarget Target_240_2:=[[73.075,133.702,0],[0.726314069,0.009187373,0.687236181,-0.009481395],[-2,0,-1,0],[9E+09,9E+09,9E+09,9E+09,9E+09,9E+09]];
    CONST robtarget Target_250_2:=[[74.399,133.623,0],[0.726314069,0.009187373,0.687236181,-0.009481395],[-2,0,-1,0],[9E+09,9E+09,9E+09,9E+09,9E+09,9E+09]];
    CONST robtarget Target_260_2:=[[76.16,133.399,0],[0.726314069,0.009187373,0.687236181,-0.009481395],[-2,0,-1,0],[9E+09,9E+09,9E+09,9E+09,9E+09,9E+09]];
    CONST robtarget Target_270_2:=[[77.475,133.111,0],[0.726314069,0.009187373,0.687236181,-0.009481395],[-2,0,-1,0],[9E+09,9E+09,9E+09,9E+09,9E+09,9E+09]];
    CONST robtarget Target_280_2:=[[78.922,132.618,0],[0.726314069,0.009187373,0.687236181,-0.009481395],[-2,0,-1,0],[9E+09,9E+09,9E+09,9E+09,9E+09,9E+09]];
    CONST robtarget Target_290_2:=[[80.057,132.032,0],[0.726314069,0.009187373,0.687236181,-0.009481395],[-2,0,-1,0],[9E+09,9E+09,9E+09,9E+09,9E+09,9E+09]];
    CONST robtarget Target_300_2:=[[81.155,131.169,0],[0.726314069,0.009187373,0.687236181,-0.009481395],[-2,0,-1,0],[9E+09,9E+09,9E+09,9E+09,9E+09,9E+09]];
    CONST robtarget Target_310_2:=[[81.768,130.466,0],[0.726314069,0.009187373,0.687236181,-0.009481395],[-2,0,-1,0],[9E+09,9E+09,9E+09,9E+09,9E+09,9E+09]];
    CONST robtarget Target_320_2:=[[82.441,129.318,0],[0.726314069,0.009187373,0.687236181,-0.009481395],[-2,0,-1,0],[9E+09,9E+09,9E+09,9E+09,9E+09,9E+09]];
    CONST robtarget Target_330_2:=[[82.754,128.475,0],[0.726314069,0.009187373,0.687236181,-0.009481395],[-2,0,-1,0],[9E+09,9E+09,9E+09,9E+09,9E+09,9E+09]];
    CONST robtarget Target_340_2:=[[82.989,127.436,0],[0.726314069,0.009187373,0.687236181,-0.009481395],[-2,0,-1,0],[9E+09,9E+09,9E+09,9E+09,9E+09,9E+09]];
    CONST robtarget Target_350_2:=[[83.108,125.846,0],[0.726314069,0.009187373,0.687236181,-0.009481395],[-2,0,-1,0],[9E+09,9E+09,9E+09,9E+09,9E+09,9E+09]];
    CONST robtarget Target_360_2:=[[83.108,110.457,0],[0.726314069,0.009187373,0.687236181,-0.009481395],[-2,0,-1,0],[9E+09,9E+09,9E+09,9E+09,9E+09,9E+09]];
    CONST robtarget Target_370_2:=[[76.106,110.457,0],[0.726314069,0.009187373,0.687236181,-0.009481395],[-2,0,-1,0],[9E+09,9E+09,9E+09,9E+09,9E+09,9E+09]];
    CONST robtarget Target_380_2:=[[76.106,112.863,0],[0.726314069,0.009187373,0.687236181,-0.009481395],[-2,0,-1,0],[9E+09,9E+09,9E+09,9E+09,9E+09,9E+09]];
    CONST robtarget Target_390_2:=[[73.262,110.797,0],[0.726314069,0.009187373,0.687236181,-0.009481395],[-2,0,-1,0],[9E+09,9E+09,9E+09,9E+09,9E+09,9E+09]];
    CONST robtarget Target_400_2:=[[68.91,109.849,0],[0.726314069,0.009187373,0.687236181,-0.009481395],[-2,0,-1,0],[9E+09,9E+09,9E+09,9E+09,9E+09,9E+09]];
    CONST robtarget Target_410_2:=[[67.809,109.921,0],[0.726314069,0.009187373,0.687236181,-0.009481395],[-2,0,-1,0],[9E+09,9E+09,9E+09,9E+09,9E+09,9E+09]];
    CONST robtarget Target_420_2:=[[66.698,110.161,0],[0.726314069,0.009187373,0.687236181,-0.009481395],[-2,0,-1,0],[9E+09,9E+09,9E+09,9E+09,9E+09,9E+09]];
    CONST robtarget Target_430_2:=[[65.802,110.508,0],[0.726314069,0.009187373,0.687236181,-0.009481395],[-2,0,-1,0],[9E+09,9E+09,9E+09,9E+09,9E+09,9E+09]];
    CONST robtarget Target_440_2:=[[64.811,111.094,0],[0.726314069,0.009187373,0.687236181,-0.009481395],[-2,0,-1,0],[9E+09,9E+09,9E+09,9E+09,9E+09,9E+09]];
    CONST robtarget Target_450_2:=[[63.886,111.896,0],[0.726314069,0.009187373,0.687236181,-0.009481395],[-2,0,-1,0],[9E+09,9E+09,9E+09,9E+09,9E+09,9E+09]];
    CONST robtarget Target_460_2:=[[63.01,112.999,0],[0.726314069,0.009187373,0.687236181,-0.009481395],[-2,0,-1,0],[9E+09,9E+09,9E+09,9E+09,9E+09,9E+09]];
    CONST robtarget Target_470_2:=[[62.505,113.958,0],[0.726314069,0.009187373,0.687236181,-0.009481395],[-2,0,-1,0],[9E+09,9E+09,9E+09,9E+09,9E+09,9E+09]];
    CONST robtarget Target_480_2:=[[62.106,115.23,0],[0.726314069,0.009187373,0.687236181,-0.009481395],[-2,0,-1,0],[9E+09,9E+09,9E+09,9E+09,9E+09,9E+09]];
    CONST robtarget Target_490_2:=[[61.935,116.747,0],[0.726314069,0.009187373,0.687236181,-0.009481395],[-2,0,-1,0],[9E+09,9E+09,9E+09,9E+09,9E+09,9E+09]];
    CONST robtarget Target_500_2:=[[61.956,117.693,0],[0.726314069,0.009187373,0.687236181,-0.009481395],[-2,0,-1,0],[9E+09,9E+09,9E+09,9E+09,9E+09,9E+09]];
    CONST robtarget Target_510_2:=[[62.24,119.422,0],[0.726314069,0.009187373,0.687236181,-0.009481395],[-2,0,-1,0],[9E+09,9E+09,9E+09,9E+09,9E+09,9E+09]];
    CONST robtarget Target_520_2:=[[62.681,120.558,0],[0.726314069,0.009187373,0.687236181,-0.009481395],[-2,0,-1,0],[9E+09,9E+09,9E+09,9E+09,9E+09,9E+09]];
    CONST robtarget Target_530_2:=[[63.326,121.537,0],[0.726314069,0.009187373,0.687236181,-0.009481395],[-2,0,-1,0],[9E+09,9E+09,9E+09,9E+09,9E+09,9E+09]];
    CONST robtarget Target_540_2:=[[64.156,122.386,0],[0.726314069,0.009187373,0.687236181,-0.009481395],[-2,0,-1,0],[9E+09,9E+09,9E+09,9E+09,9E+09,9E+09]];
    CONST robtarget Target_550_2:=[[65.088,123.055,0],[0.726314069,0.009187373,0.687236181,-0.009481395],[-2,0,-1,0],[9E+09,9E+09,9E+09,9E+09,9E+09,9E+09]];
    CONST robtarget Target_560_2:=[[65.847,123.463,0],[0.726314069,0.009187373,0.687236181,-0.009481395],[-2,0,-1,0],[9E+09,9E+09,9E+09,9E+09,9E+09,9E+09]];
    CONST robtarget Target_570_2:=[[69.214,124.548,0],[0.726314069,0.009187373,0.687236181,-0.009481395],[-2,0,-1,0],[9E+09,9E+09,9E+09,9E+09,9E+09,9E+09]];
    CONST robtarget Target_580_2:=[[70.751,124.795,0],[0.726314069,0.009187373,0.687236181,-0.009481395],[-2,0,-1,0],[9E+09,9E+09,9E+09,9E+09,9E+09,9E+09]];
    CONST robtarget Target_590_2:=[[72.603,125.014,0],[0.726314069,0.009187373,0.687236181,-0.009481395],[-2,0,-1,0],[9E+09,9E+09,9E+09,9E+09,9E+09,9E+09]];
    CONST robtarget Target_600_2:=[[74.414,125.184,0],[0.726314069,0.009187373,0.687236181,-0.009481395],[-2,0,-1,0],[9E+09,9E+09,9E+09,9E+09,9E+09,9E+09]];
    CONST robtarget Target_610_2:=[[76.155,125.311,0],[0.726314069,0.009187373,0.687236181,-0.009481395],[-2,0,-1,0],[9E+09,9E+09,9E+09,9E+09,9E+09,9E+09]];
    CONST robtarget Target_620_2:=[[76.155,125.432,0],[0.726314069,0.009187373,0.687236181,-0.009481395],[-2,0,-1,0],[9E+09,9E+09,9E+09,9E+09,9E+09,9E+09]];
    CONST robtarget Target_630_2:=[[76.114,126.039,0],[0.726314069,0.009187373,0.687236181,-0.009481395],[-2,0,-1,0],[9E+09,9E+09,9E+09,9E+09,9E+09,9E+09]];
    CONST robtarget Target_640_2:=[[75.849,126.936,0],[0.726314069,0.009187373,0.687236181,-0.009481395],[-2,0,-1,0],[9E+09,9E+09,9E+09,9E+09,9E+09,9E+09]];
    CONST robtarget Target_650_2:=[[75.219,127.729,0],[0.726314069,0.009187373,0.687236181,-0.009481395],[-2,0,-1,0],[9E+09,9E+09,9E+09,9E+09,9E+09,9E+09]];
    CONST robtarget Target_660_2:=[[74.486,128.154,0],[0.726314069,0.009187373,0.687236181,-0.009481395],[-2,0,-1,0],[9E+09,9E+09,9E+09,9E+09,9E+09,9E+09]];
    CONST robtarget Target_670_2:=[[73.351,128.499,0],[0.726314069,0.009187373,0.687236181,-0.009481395],[-2,0,-1,0],[9E+09,9E+09,9E+09,9E+09,9E+09,9E+09]];
    CONST robtarget Target_680_2:=[[72.285,128.661,0],[0.726314069,0.009187373,0.687236181,-0.009481395],[-2,0,-1,0],[9E+09,9E+09,9E+09,9E+09,9E+09,9E+09]];
    CONST robtarget Target_690_2:=[[71.471,128.72,0],[0.726314069,0.009187373,0.687236181,-0.009481395],[-2,0,-1,0],[9E+09,9E+09,9E+09,9E+09,9E+09,9E+09]];
    CONST robtarget Target_700_2:=[[70.612,128.739,0],[0.726314069,0.009187373,0.687236181,-0.009481395],[-2,0,-1,0],[9E+09,9E+09,9E+09,9E+09,9E+09,9E+09]];
    CONST robtarget Target_710_2:=[[64.437,127.134,0],[0.726314069,0.009187373,0.687236181,-0.009481395],[-2,0,-1,0],[9E+09,9E+09,9E+09,9E+09,9E+09,9E+09]];
    CONST robtarget Target_720_2:=[[63.829,127.134,0],[0.726314069,0.009187373,0.687236181,-0.009481395],[-2,0,-1,0],[9E+09,9E+09,9E+09,9E+09,9E+09,9E+09]];
    CONST robtarget Target_730_2:=[[63.829,132.604,0],[0.726314069,0.009187373,0.687236181,-0.009481395],[-2,0,-1,0],[9E+09,9E+09,9E+09,9E+09,9E+09,9E+09]];
    CONST robtarget Target_740_2:=[[63.829,132.604,10],[0.726314069,0.009187373,0.687236181,-0.009481395],[-2,0,-1,0],[9E+09,9E+09,9E+09,9E+09,9E+09,9E+09]];
    CONST robtarget Target_750_2:=[[76.106,121.056,10],[0.726314069,0.009187373,0.687236181,-0.009481395],[-2,0,-1,0],[9E+09,9E+09,9E+09,9E+09,9E+09,9E+09]];
    CONST robtarget Target_760_2:=[[76.106,121.056,0],[0.726314069,0.009187373,0.687236181,-0.009481395],[-2,0,-1,0],[9E+09,9E+09,9E+09,9E+09,9E+09,9E+09]];
    CONST robtarget Target_770_2:=[[71.025,120.23,0],[0.726314069,0.009187373,0.687236181,-0.009481395],[-2,0,-1,0],[9E+09,9E+09,9E+09,9E+09,9E+09,9E+09]];
    CONST robtarget Target_780_2:=[[70.06,119.739,0],[0.726314069,0.009187373,0.687236181,-0.009481395],[-2,0,-1,0],[9E+09,9E+09,9E+09,9E+09,9E+09,9E+09]];
    CONST robtarget Target_790_2:=[[69.338,118.892,0],[0.726314069,0.009187373,0.687236181,-0.009481395],[-2,0,-1,0],[9E+09,9E+09,9E+09,9E+09,9E+09,9E+09]];
    CONST robtarget Target_800_2:=[[69.114,118.205,0],[0.726314069,0.009187373,0.687236181,-0.009481395],[-2,0,-1,0],[9E+09,9E+09,9E+09,9E+09,9E+09,9E+09]];
    CONST robtarget Target_810_2:=[[69.056,117.55,0],[0.726314069,0.009187373,0.687236181,-0.009481395],[-2,0,-1,0],[9E+09,9E+09,9E+09,9E+09,9E+09,9E+09]];
    CONST robtarget Target_820_2:=[[69.091,116.93,0],[0.726314069,0.009187373,0.687236181,-0.009481395],[-2,0,-1,0],[9E+09,9E+09,9E+09,9E+09,9E+09,9E+09]];
    CONST robtarget Target_830_2:=[[69.292,116.148,0],[0.726314069,0.009187373,0.687236181,-0.009481395],[-2,0,-1,0],[9E+09,9E+09,9E+09,9E+09,9E+09,9E+09]];
    CONST robtarget Target_840_2:=[[69.919,115.356,0],[0.726314069,0.009187373,0.687236181,-0.009481395],[-2,0,-1,0],[9E+09,9E+09,9E+09,9E+09,9E+09,9E+09]];
    CONST robtarget Target_850_2:=[[70.774,114.964,0],[0.726314069,0.009187373,0.687236181,-0.009481395],[-2,0,-1,0],[9E+09,9E+09,9E+09,9E+09,9E+09,9E+09]];
    CONST robtarget Target_860_2:=[[71.742,114.79,0],[0.726314069,0.009187373,0.687236181,-0.009481395],[-2,0,-1,0],[9E+09,9E+09,9E+09,9E+09,9E+09,9E+09]];
    CONST robtarget Target_870_2:=[[72.46,114.76,0],[0.726314069,0.009187373,0.687236181,-0.009481395],[-2,0,-1,0],[9E+09,9E+09,9E+09,9E+09,9E+09,9E+09]];
    CONST robtarget Target_880_2:=[[72.459,114.76,0],[0.726314069,0.009187373,0.687236181,-0.009481395],[-2,0,-1,0],[9E+09,9E+09,9E+09,9E+09,9E+09,9E+09]];
    CONST robtarget Target_890_2:=[[73.597,114.916,0],[0.726314069,0.009187373,0.687236181,-0.009481395],[-2,0,-1,0],[9E+09,9E+09,9E+09,9E+09,9E+09,9E+09]];
    CONST robtarget Target_900_2:=[[74.622,115.309,0],[0.726314069,0.009187373,0.687236181,-0.009481395],[-2,0,-1,0],[9E+09,9E+09,9E+09,9E+09,9E+09,9E+09]];
    CONST robtarget Target_910_2:=[[75.105,115.58,0],[0.726314069,0.009187373,0.687236181,-0.009481395],[-2,0,-1,0],[9E+09,9E+09,9E+09,9E+09,9E+09,9E+09]];
    CONST robtarget Target_920_2:=[[75.771,116.063,0],[0.726314069,0.009187373,0.687236181,-0.009481395],[-2,0,-1,0],[9E+09,9E+09,9E+09,9E+09,9E+09,9E+09]];
    CONST robtarget Target_930_2:=[[76.106,116.364,0],[0.726314069,0.009187373,0.687236181,-0.009481395],[-2,0,-1,0],[9E+09,9E+09,9E+09,9E+09,9E+09,9E+09]];
    CONST robtarget Target_940_2:=[[76.106,121.056,0],[0.726314069,0.009187373,0.687236181,-0.009481395],[-2,0,-1,0],[9E+09,9E+09,9E+09,9E+09,9E+09,9E+09]];
    CONST robtarget Target_950_2:=[[76.106,121.056,10],[0.726314069,0.009187373,0.687236181,-0.009481395],[-2,0,-1,0],[9E+09,9E+09,9E+09,9E+09,9E+09,9E+09]];
    CONST robtarget Target_960_2:=[[86.049,133.09,10],[0.726314069,0.009187373,0.687236181,-0.009481395],[-1,0,-1,0],[9E+09,9E+09,9E+09,9E+09,9E+09,9E+09]];
    CONST robtarget Target_970_2:=[[86.049,133.09,0],[0.726314069,0.009187373,0.687236181,-0.009481395],[-1,0,-1,0],[9E+09,9E+09,9E+09,9E+09,9E+09,9E+09]];
    CONST robtarget Target_980_2:=[[88.87,133.09,0],[0.726314069,0.009187373,0.687236181,-0.009481395],[-1,0,-1,0],[9E+09,9E+09,9E+09,9E+09,9E+09,9E+09]];
    CONST robtarget Target_990_2:=[[88.87,133.722,0],[0.726314069,0.009187373,0.687236181,-0.009481395],[-1,0,-1,0],[9E+09,9E+09,9E+09,9E+09,9E+09,9E+09]];
    CONST robtarget Target_1000_2:=[[88.943,135.17,0],[0.726314069,0.009187373,0.687236181,-0.009481395],[-1,0,-1,0],[9E+09,9E+09,9E+09,9E+09,9E+09,9E+09]];
    CONST robtarget Target_1010_2:=[[89.33,137.086,0],[0.726314069,0.009187373,0.687236181,-0.009481395],[-1,0,-1,0],[9E+09,9E+09,9E+09,9E+09,9E+09,9E+09]];
    CONST robtarget Target_1020_2:=[[90.035,138.666,0],[0.726314069,0.009187373,0.687236181,-0.009481395],[-1,0,-1,0],[9E+09,9E+09,9E+09,9E+09,9E+09,9E+09]];
    CONST robtarget Target_1030_2:=[[90.843,139.72,0],[0.726314069,0.009187373,0.687236181,-0.009481395],[-1,0,-1,0],[9E+09,9E+09,9E+09,9E+09,9E+09,9E+09]];
    CONST robtarget Target_1040_2:=[[92.423,140.908,0],[0.726314069,0.009187373,0.687236181,-0.009481395],[-1,0,-1,0],[9E+09,9E+09,9E+09,9E+09,9E+09,9E+09]];
    CONST robtarget Target_1050_2:=[[94.644,141.698,0],[0.726314069,0.009187373,0.687236181,-0.009481395],[-1,0,-1,0],[9E+09,9E+09,9E+09,9E+09,9E+09,9E+09]];
    CONST robtarget Target_1060_2:=[[96.483,141.95,0],[0.726314069,0.009187373,0.687236181,-0.009481395],[-1,-1,-1,0],[9E+09,9E+09,9E+09,9E+09,9E+09,9E+09]];
    CONST robtarget Target_1070_2:=[[97.646,141.988,0],[0.726314069,0.009187373,0.687236181,-0.009481395],[-1,-1,0,0],[9E+09,9E+09,9E+09,9E+09,9E+09,9E+09]];
    CONST robtarget Target_1080_2:=[[102.8,141.575,0],[0.726314069,0.009187373,0.687236181,-0.009481395],[-1,-1,0,0],[9E+09,9E+09,9E+09,9E+09,9E+09,9E+09]];
    CONST robtarget Target_1090_2:=[[102.8,136.47,0],[0.726314069,0.009187373,0.687236181,-0.009481395],[-1,-1,0,0],[9E+09,9E+09,9E+09,9E+09,9E+09,9E+09]];
    CONST robtarget Target_1100_2:=[[102.265,136.47,0],[0.726314069,0.009187373,0.687236181,-0.009481395],[-1,-1,0,0],[9E+09,9E+09,9E+09,9E+09,9E+09,9E+09]];
    CONST robtarget Target_1110_2:=[[99.372,136.98,0],[0.726314069,0.009187373,0.687236181,-0.009481395],[-1,-1,0,0],[9E+09,9E+09,9E+09,9E+09,9E+09,9E+09]];
    CONST robtarget Target_1120_2:=[[98.552,136.947,0],[0.726314069,0.009187373,0.687236181,-0.009481395],[-1,-1,0,0],[9E+09,9E+09,9E+09,9E+09,9E+09,9E+09]];
    CONST robtarget Target_1130_2:=[[97.623,136.799,0],[0.726314069,0.009187373,0.687236181,-0.009481395],[-1,-1,0,0],[9E+09,9E+09,9E+09,9E+09,9E+09,9E+09]];
    CONST robtarget Target_1140_2:=[[96.675,136.388,0],[0.726314069,0.009187373,0.687236181,-0.009481395],[-1,-1,0,0],[9E+09,9E+09,9E+09,9E+09,9E+09,9E+09]];
    CONST robtarget Target_1150_2:=[[96.077,135.652,0],[0.726314069,0.009187373,0.687236181,-0.009481395],[-1,0,-1,0],[9E+09,9E+09,9E+09,9E+09,9E+09,9E+09]];
    CONST robtarget Target_1160_2:=[[95.864,135.05,0],[0.726314069,0.009187373,0.687236181,-0.009481395],[-1,0,-1,0],[9E+09,9E+09,9E+09,9E+09,9E+09,9E+09]];
    CONST robtarget Target_1170_2:=[[95.723,134.236,0],[0.726314069,0.009187373,0.687236181,-0.009481395],[-1,0,-1,0],[9E+09,9E+09,9E+09,9E+09,9E+09,9E+09]];
    CONST robtarget Target_1180_2:=[[95.677,133.26,0],[0.726314069,0.009187373,0.687236181,-0.009481395],[-1,0,-1,0],[9E+09,9E+09,9E+09,9E+09,9E+09,9E+09]];
    CONST robtarget Target_1190_2:=[[95.677,133.09,0],[0.726314069,0.009187373,0.687236181,-0.009481395],[-1,0,-1,0],[9E+09,9E+09,9E+09,9E+09,9E+09,9E+09]];
    CONST robtarget Target_1200_2:=[[101.293,133.09,0],[0.726314069,0.009187373,0.687236181,-0.009481395],[-1,-1,0,0],[9E+09,9E+09,9E+09,9E+09,9E+09,9E+09]];
    CONST robtarget Target_1210_2:=[[101.293,128.179,0],[0.726314069,0.009187373,0.687236181,-0.009481395],[-1,-1,0,0],[9E+09,9E+09,9E+09,9E+09,9E+09,9E+09]];
    CONST robtarget Target_1220_2:=[[95.92,128.179,0],[0.726314069,0.009187373,0.687236181,-0.009481395],[-1,0,-1,0],[9E+09,9E+09,9E+09,9E+09,9E+09,9E+09]];
    CONST robtarget Target_1230_2:=[[95.92,110.457,0],[0.726314069,0.009187373,0.687236181,-0.009481395],[-1,0,-1,0],[9E+09,9E+09,9E+09,9E+09,9E+09,9E+09]];
    CONST robtarget Target_1240_2:=[[88.87,110.457,0],[0.726314069,0.009187373,0.687236181,-0.009481395],[-1,0,-1,0],[9E+09,9E+09,9E+09,9E+09,9E+09,9E+09]];
    CONST robtarget Target_1250_2:=[[88.87,128.179,0],[0.726314069,0.009187373,0.687236181,-0.009481395],[-1,0,-1,0],[9E+09,9E+09,9E+09,9E+09,9E+09,9E+09]];
    CONST robtarget Target_1260_2:=[[86.049,128.179,0],[0.726314069,0.009187373,0.687236181,-0.009481395],[-1,0,-1,0],[9E+09,9E+09,9E+09,9E+09,9E+09,9E+09]];
    CONST robtarget Target_1270_2:=[[86.049,133.09,0],[0.726314069,0.009187373,0.687236181,-0.009481395],[-1,0,-1,0],[9E+09,9E+09,9E+09,9E+09,9E+09,9E+09]];
    CONST robtarget Target_1280_2:=[[86.049,133.09,10],[0.726314069,0.009187373,0.687236181,-0.009481395],[-1,0,-1,0],[9E+09,9E+09,9E+09,9E+09,9E+09,9E+09]];
    CONST robtarget Target_1290_2:=[[109.485,124.679,10],[0.726314069,0.009187373,0.687236181,-0.009481395],[-1,-1,0,0],[9E+09,9E+09,9E+09,9E+09,9E+09,9E+09]];
    CONST robtarget Target_1300_2:=[[109.485,124.679,0],[0.726314069,0.009187373,0.687236181,-0.009481395],[-1,-1,0,0],[9E+09,9E+09,9E+09,9E+09,9E+09,9E+09]];
    CONST robtarget Target_1310_2:=[[109.701,126.061,0],[0.726314069,0.009187373,0.687236181,-0.009481395],[-1,-1,0,0],[9E+09,9E+09,9E+09,9E+09,9E+09,9E+09]];
    CONST robtarget Target_1320_2:=[[110.324,127.465,0],[0.726314069,0.009187373,0.687236181,-0.009481395],[-1,-1,0,0],[9E+09,9E+09,9E+09,9E+09,9E+09,9E+09]];
    CONST robtarget Target_1330_2:=[[111.27,128.475,0],[0.726314069,0.009187373,0.687236181,-0.009481395],[-1,-1,0,0],[9E+09,9E+09,9E+09,9E+09,9E+09,9E+09]];
    CONST robtarget Target_1340_2:=[[112.867,129.166,0],[0.726314069,0.009187373,0.687236181,-0.009481395],[-1,-1,0,0],[9E+09,9E+09,9E+09,9E+09,9E+09,9E+09]];
    CONST robtarget Target_1350_2:=[[114.033,129.273,0],[0.726314069,0.009187373,0.687236181,-0.009481395],[-1,-1,0,0],[9E+09,9E+09,9E+09,9E+09,9E+09,9E+09]];
    CONST robtarget Target_1360_2:=[[114.895,129.209,0],[0.726314069,0.009187373,0.687236181,-0.009481395],[-1,-1,0,0],[9E+09,9E+09,9E+09,9E+09,9E+09,9E+09]];
    CONST robtarget Target_1370_2:=[[116.013,128.871,0],[0.726314069,0.009187373,0.687236181,-0.009481395],[-1,-1,0,0],[9E+09,9E+09,9E+09,9E+09,9E+09,9E+09]];
    CONST robtarget Target_1380_2:=[[116.864,128.257,0],[0.726314069,0.009187373,0.687236181,-0.009481395],[-1,-1,0,0],[9E+09,9E+09,9E+09,9E+09,9E+09,9E+09]];
    CONST robtarget Target_1390_2:=[[117.585,127.137,0],[0.726314069,0.009187373,0.687236181,-0.009481395],[-1,-1,0,0],[9E+09,9E+09,9E+09,9E+09,9E+09,9E+09]];
    CONST robtarget Target_1400_2:=[[117.862,126.264,0],[0.726314069,0.009187373,0.687236181,-0.009481395],[-1,-1,0,0],[9E+09,9E+09,9E+09,9E+09,9E+09,9E+09]];
    CONST robtarget Target_1410_2:=[[118,125.407,0],[0.726314069,0.009187373,0.687236181,-0.009481395],[-1,-1,0,0],[9E+09,9E+09,9E+09,9E+09,9E+09,9E+09]];
    CONST robtarget Target_1420_2:=[[118.043,124.679,0],[0.726314069,0.009187373,0.687236181,-0.009481395],[-1,-1,0,0],[9E+09,9E+09,9E+09,9E+09,9E+09,9E+09]];
    CONST robtarget Target_1430_2:=[[109.485,124.679,0],[0.726314069,0.009187373,0.687236181,-0.009481395],[-1,-1,0,0],[9E+09,9E+09,9E+09,9E+09,9E+09,9E+09]];
    CONST robtarget Target_1440_2:=[[109.485,124.679,10],[0.726314069,0.009187373,0.687236181,-0.009481395],[-1,-1,0,0],[9E+09,9E+09,9E+09,9E+09,9E+09,9E+09]];
    CONST robtarget Target_1450_2:=[[124.996,120.424,10],[0.726314069,0.009187373,0.687236181,-0.009481395],[-1,-1,0,0],[9E+09,9E+09,9E+09,9E+09,9E+09,9E+09]];
    CONST robtarget Target_1460_2:=[[124.996,120.424,0],[0.726314069,0.009187373,0.687236181,-0.009481395],[-1,-1,0,0],[9E+09,9E+09,9E+09,9E+09,9E+09,9E+09]];
    CONST robtarget Target_1470_2:=[[109.51,120.424,0],[0.726314069,0.009187373,0.687236181,-0.009481395],[-1,-1,0,0],[9E+09,9E+09,9E+09,9E+09,9E+09,9E+09]];
    CONST robtarget Target_1480_2:=[[110.356,117.497,0],[0.726314069,0.009187373,0.687236181,-0.009481395],[-1,-1,0,0],[9E+09,9E+09,9E+09,9E+09,9E+09,9E+09]];
    CONST robtarget Target_1490_2:=[[111.754,116.065,0],[0.726314069,0.009187373,0.687236181,-0.009481395],[-1,-1,0,0],[9E+09,9E+09,9E+09,9E+09,9E+09,9E+09]];
    CONST robtarget Target_1500_2:=[[113.375,115.326,0],[0.726314069,0.009187373,0.687236181,-0.009481395],[-1,-1,0,0],[9E+09,9E+09,9E+09,9E+09,9E+09,9E+09]];
    CONST robtarget Target_1510_2:=[[115.333,114.996,0],[0.726314069,0.009187373,0.687236181,-0.009481395],[-1,-1,0,0],[9E+09,9E+09,9E+09,9E+09,9E+09,9E+09]];
    CONST robtarget Target_1520_2:=[[117.175,114.979,0],[0.726314069,0.009187373,0.687236181,-0.009481395],[-1,-1,0,0],[9E+09,9E+09,9E+09,9E+09,9E+09,9E+09]];
    CONST robtarget Target_1530_2:=[[118.717,115.194,0],[0.726314069,0.009187373,0.687236181,-0.009481395],[-1,-1,0,0],[9E+09,9E+09,9E+09,9E+09,9E+09,9E+09]];
    CONST robtarget Target_1540_2:=[[120.709,115.808,0],[0.726314069,0.009187373,0.687236181,-0.009481395],[-1,-1,0,0],[9E+09,9E+09,9E+09,9E+09,9E+09,9E+09]];
    CONST robtarget Target_1550_2:=[[121.033,115.951,0],[0.726314069,0.009187373,0.687236181,-0.009481395],[-1,-1,0,0],[9E+09,9E+09,9E+09,9E+09,9E+09,9E+09]];
    CONST robtarget Target_1560_2:=[[123.829,117.555,0],[0.726314069,0.009187373,0.687236181,-0.009481395],[-1,-1,0,0],[9E+09,9E+09,9E+09,9E+09,9E+09,9E+09]];
    CONST robtarget Target_1570_2:=[[124.583,117.555,0],[0.726314069,0.009187373,0.687236181,-0.009481395],[-1,-1,0,0],[9E+09,9E+09,9E+09,9E+09,9E+09,9E+09]];
    CONST robtarget Target_1580_2:=[[124.583,111.721,0],[0.726314069,0.009187373,0.687236181,-0.009481395],[-1,-1,0,0],[9E+09,9E+09,9E+09,9E+09,9E+09,9E+09]];
    CONST robtarget Target_1590_2:=[[121.033,110.505,0],[0.726314069,0.009187373,0.687236181,-0.009481395],[-1,-1,0,0],[9E+09,9E+09,9E+09,9E+09,9E+09,9E+09]];
    CONST robtarget Target_1600_2:=[[115.709,109.849,0],[0.726314069,0.009187373,0.687236181,-0.009481395],[-1,-1,0,0],[9E+09,9E+09,9E+09,9E+09,9E+09,9E+09]];
    CONST robtarget Target_1610_2:=[[113.106,109.988,0],[0.726314069,0.009187373,0.687236181,-0.009481395],[-1,-1,0,0],[9E+09,9E+09,9E+09,9E+09,9E+09,9E+09]];
    CONST robtarget Target_1620_2:=[[110.207,110.564,0],[0.726314069,0.009187373,0.687236181,-0.009481395],[-1,-1,0,0],[9E+09,9E+09,9E+09,9E+09,9E+09,9E+09]];
    CONST robtarget Target_1630_2:=[[108.088,111.404,0],[0.726314069,0.009187373,0.687236181,-0.009481395],[-1,-1,0,0],[9E+09,9E+09,9E+09,9E+09,9E+09,9E+09]];
    CONST robtarget Target_1640_2:=[[106.39,112.481,0],[0.726314069,0.009187373,0.687236181,-0.009481395],[-1,-1,0,0],[9E+09,9E+09,9E+09,9E+09,9E+09,9E+09]];
    CONST robtarget Target_1650_2:=[[105.004,113.799,0],[0.726314069,0.009187373,0.687236181,-0.009481395],[-1,-1,0,0],[9E+09,9E+09,9E+09,9E+09,9E+09,9E+09]];
    CONST robtarget Target_1660_2:=[[103.854,115.462,0],[0.726314069,0.009187373,0.687236181,-0.009481395],[-1,-1,0,0],[9E+09,9E+09,9E+09,9E+09,9E+09,9E+09]];
    CONST robtarget Target_1670_2:=[[103.1,117.221,0],[0.726314069,0.009187373,0.687236181,-0.009481395],[-1,-1,0,0],[9E+09,9E+09,9E+09,9E+09,9E+09,9E+09]];
    CONST robtarget Target_1680_2:=[[102.678,118.94,0],[0.726314069,0.009187373,0.687236181,-0.009481395],[-1,-1,0,0],[9E+09,9E+09,9E+09,9E+09,9E+09,9E+09]];
    CONST robtarget Target_1690_2:=[[102.466,121.144,0],[0.726314069,0.009187373,0.687236181,-0.009481395],[-1,-1,0,0],[9E+09,9E+09,9E+09,9E+09,9E+09,9E+09]];
    CONST robtarget Target_1700_2:=[[102.503,122.901,0],[0.726314069,0.009187373,0.687236181,-0.009481395],[-1,-1,0,0],[9E+09,9E+09,9E+09,9E+09,9E+09,9E+09]];
    CONST robtarget Target_1710_2:=[[102.895,125.435,0],[0.726314069,0.009187373,0.687236181,-0.009481395],[-1,-1,0,0],[9E+09,9E+09,9E+09,9E+09,9E+09,9E+09]];
    CONST robtarget Target_1720_2:=[[103.544,127.348,0],[0.726314069,0.009187373,0.687236181,-0.009481395],[-1,-1,0,0],[9E+09,9E+09,9E+09,9E+09,9E+09,9E+09]];
    CONST robtarget Target_1730_2:=[[104.846,129.56,0],[0.726314069,0.009187373,0.687236181,-0.009481395],[-1,-1,0,0],[9E+09,9E+09,9E+09,9E+09,9E+09,9E+09]];
    CONST robtarget Target_1740_2:=[[107.173,131.787,0],[0.726314069,0.009187373,0.687236181,-0.009481395],[-1,-1,0,0],[9E+09,9E+09,9E+09,9E+09,9E+09,9E+09]];
    CONST robtarget Target_1750_2:=[[110.252,133.228,0],[0.726314069,0.009187373,0.687236181,-0.009481395],[-1,-1,0,0],[9E+09,9E+09,9E+09,9E+09,9E+09,9E+09]];
    CONST robtarget Target_1760_2:=[[112.653,133.696,0],[0.726314069,0.009187373,0.687236181,-0.009481395],[-1,-1,0,0],[9E+09,9E+09,9E+09,9E+09,9E+09,9E+09]];
    CONST robtarget Target_1770_2:=[[115.907,133.745,0],[0.726314069,0.009187373,0.687236181,-0.009481395],[-1,-1,0,0],[9E+09,9E+09,9E+09,9E+09,9E+09,9E+09]];
    CONST robtarget Target_1780_2:=[[118.059,133.408,0],[0.726314069,0.009187373,0.687236181,-0.009481395],[-1,-1,0,0],[9E+09,9E+09,9E+09,9E+09,9E+09,9E+09]];
    CONST robtarget Target_1790_2:=[[120.042,132.698,0],[0.726314069,0.009187373,0.687236181,-0.009481395],[-1,-1,0,0],[9E+09,9E+09,9E+09,9E+09,9E+09,9E+09]];
    CONST robtarget Target_1800_2:=[[121.361,131.894,0],[0.726314069,0.009187373,0.687236181,-0.009481395],[-1,-1,0,0],[9E+09,9E+09,9E+09,9E+09,9E+09,9E+09]];
    CONST robtarget Target_1810_2:=[[122.662,130.659,0],[0.726314069,0.009187373,0.687236181,-0.009481395],[-1,-1,0,0],[9E+09,9E+09,9E+09,9E+09,9E+09,9E+09]];
    CONST robtarget Target_1820_2:=[[123.82,128.868,0],[0.726314069,0.009187373,0.687236181,-0.009481395],[-1,-1,0,0],[9E+09,9E+09,9E+09,9E+09,9E+09,9E+09]];
    CONST robtarget Target_1830_2:=[[124.578,126.747,0],[0.726314069,0.009187373,0.687236181,-0.009481395],[-1,-1,0,0],[9E+09,9E+09,9E+09,9E+09,9E+09,9E+09]];
    CONST robtarget Target_1840_2:=[[124.955,124.236,0],[0.726314069,0.009187373,0.687236181,-0.009481395],[-1,-1,0,0],[9E+09,9E+09,9E+09,9E+09,9E+09,9E+09]];
    CONST robtarget Target_1850_2:=[[124.996,122.121,0],[0.726314069,0.009187373,0.687236181,-0.009481395],[-1,-1,0,0],[9E+09,9E+09,9E+09,9E+09,9E+09,9E+09]];
    CONST robtarget Target_1860_2:=[[124.996,120.424,0],[0.726314069,0.009187373,0.687236181,-0.009481395],[-1,-1,0,0],[9E+09,9E+09,9E+09,9E+09,9E+09,9E+09]];
    CONST robtarget Target_1870_2:=[[124.996,120.424,10],[0.726314069,0.009187373,0.687236181,-0.009481395],[-1,-1,0,0],[9E+09,9E+09,9E+09,9E+09,9E+09,9E+09]];
    CONST robtarget Target_1880_2:=[[48.093,102.54,10],[0.726314069,0.009187373,0.687236181,-0.009481395],[-2,0,-1,0],[9E+09,9E+09,9E+09,9E+09,9E+09,9E+09]];
    CONST robtarget Target_1890_2:=[[48.093,102.54,0],[0.726314069,0.009187373,0.687236181,-0.009481395],[-2,0,-1,0],[9E+09,9E+09,9E+09,9E+09,9E+09,9E+09]];
    CONST robtarget Target_1900_2:=[[43.231,104.473,0],[0.726314069,0.009187373,0.687236181,-0.009481395],[-2,0,-1,0],[9E+09,9E+09,9E+09,9E+09,9E+09,9E+09]];
    CONST robtarget Target_1910_2:=[[37.105,105.19,0],[0.726314069,0.009187373,0.687236181,-0.009481395],[-2,0,-1,0],[9E+09,9E+09,9E+09,9E+09,9E+09,9E+09]];
    CONST robtarget Target_1920_2:=[[32.913,104.788,0],[0.726314069,0.009187373,0.687236181,-0.009481395],[-2,0,-1,0],[9E+09,9E+09,9E+09,9E+09,9E+09,9E+09]];
    CONST robtarget Target_1930_2:=[[30.425,104.066,0],[0.726314069,0.009187373,0.687236181,-0.009481395],[-2,0,-1,0],[9E+09,9E+09,9E+09,9E+09,9E+09,9E+09]];
    CONST robtarget Target_1940_2:=[[27.453,102.491,0],[0.726314069,0.009187373,0.687236181,-0.009481395],[-2,0,-1,0],[9E+09,9E+09,9E+09,9E+09,9E+09,9E+09]];
    CONST robtarget Target_1950_2:=[[25.682,101,0],[0.726314069,0.009187373,0.687236181,-0.009481395],[-2,0,-1,0],[9E+09,9E+09,9E+09,9E+09,9E+09,9E+09]];
    CONST robtarget Target_1960_2:=[[24.18,99.225,0],[0.726314069,0.009187373,0.687236181,-0.009481395],[-2,0,-1,0],[9E+09,9E+09,9E+09,9E+09,9E+09,9E+09]];
    CONST robtarget Target_1970_2:=[[23.043,97.314,0],[0.726314069,0.009187373,0.687236181,-0.009481395],[-2,0,-1,0],[9E+09,9E+09,9E+09,9E+09,9E+09,9E+09]];
    CONST robtarget Target_1980_2:=[[22.382,95.73,0],[0.726314069,0.009187373,0.687236181,-0.009481395],[-2,0,-1,0],[9E+09,9E+09,9E+09,9E+09,9E+09,9E+09]];
    CONST robtarget Target_1990_2:=[[21.885,93.998,0],[0.726314069,0.009187373,0.687236181,-0.009481395],[-2,0,-1,0],[9E+09,9E+09,9E+09,9E+09,9E+09,9E+09]];
    CONST robtarget Target_2000_2:=[[21.534,91.845,0],[0.726314069,0.009187373,0.687236181,-0.009481395],[-2,0,-1,0],[9E+09,9E+09,9E+09,9E+09,9E+09,9E+09]];
    CONST robtarget Target_2010_2:=[[21.424,89.631,0],[0.726314069,0.009187373,0.687236181,-0.009481395],[-2,0,-1,0],[9E+09,9E+09,9E+09,9E+09,9E+09,9E+09]];
    CONST robtarget Target_2020_2:=[[21.598,86.718,0],[0.726314069,0.009187373,0.687236181,-0.009481395],[-2,0,-1,0],[9E+09,9E+09,9E+09,9E+09,9E+09,9E+09]];
    CONST robtarget Target_2030_2:=[[22.061,84.31,0],[0.726314069,0.009187373,0.687236181,-0.009481395],[-2,0,-1,0],[9E+09,9E+09,9E+09,9E+09,9E+09,9E+09]];
    CONST robtarget Target_2040_2:=[[22.438,83.089,0],[0.726314069,0.009187373,0.687236181,-0.009481395],[-2,0,-1,0],[9E+09,9E+09,9E+09,9E+09,9E+09,9E+09]];
    CONST robtarget Target_2050_2:=[[23.52,80.745,0],[0.726314069,0.009187373,0.687236181,-0.009481395],[-2,0,-1,0],[9E+09,9E+09,9E+09,9E+09,9E+09,9E+09]];
    CONST robtarget Target_2060_2:=[[25.622,78.054,0],[0.726314069,0.009187373,0.687236181,-0.009481395],[-2,0,-1,0],[9E+09,9E+09,9E+09,9E+09,9E+09,9E+09]];
    CONST robtarget Target_2070_2:=[[28.684,75.816,0],[0.726314069,0.009187373,0.687236181,-0.009481395],[-2,0,-1,0],[9E+09,9E+09,9E+09,9E+09,9E+09,9E+09]];
    CONST robtarget Target_2080_2:=[[31.534,74.671,0],[0.726314069,0.009187373,0.687236181,-0.009481395],[-2,0,-1,0],[9E+09,9E+09,9E+09,9E+09,9E+09,9E+09]];
    CONST robtarget Target_2090_2:=[[35.573,74.011,0],[0.726314069,0.009187373,0.687236181,-0.009481395],[-2,0,-1,0],[9E+09,9E+09,9E+09,9E+09,9E+09,9E+09]];
    CONST robtarget Target_2100_2:=[[38.167,74.008,0],[0.726314069,0.009187373,0.687236181,-0.009481395],[-2,0,-1,0],[9E+09,9E+09,9E+09,9E+09,9E+09,9E+09]];
    CONST robtarget Target_2110_2:=[[40.483,74.234,0],[0.726314069,0.009187373,0.687236181,-0.009481395],[-2,0,-1,0],[9E+09,9E+09,9E+09,9E+09,9E+09,9E+09]];
    CONST robtarget Target_2120_2:=[[43.194,74.764,0],[0.726314069,0.009187373,0.687236181,-0.009481395],[-2,0,-1,0],[9E+09,9E+09,9E+09,9E+09,9E+09,9E+09]];
    CONST robtarget Target_2130_2:=[[46.412,75.66,0],[0.726314069,0.009187373,0.687236181,-0.009481395],[-2,0,-1,0],[9E+09,9E+09,9E+09,9E+09,9E+09,9E+09]];
    CONST robtarget Target_2140_2:=[[48.215,76.308,0],[0.726314069,0.009187373,0.687236181,-0.009481395],[-2,0,-1,0],[9E+09,9E+09,9E+09,9E+09,9E+09,9E+09]];
    CONST robtarget Target_2150_2:=[[48.215,91.09,0],[0.726314069,0.009187373,0.687236181,-0.009481395],[-2,0,-1,0],[9E+09,9E+09,9E+09,9E+09,9E+09,9E+09]];
    CONST robtarget Target_2160_2:=[[35.111,91.09,0],[0.726314069,0.009187373,0.687236181,-0.009481395],[-2,0,-1,0],[9E+09,9E+09,9E+09,9E+09,9E+09,9E+09]];
    CONST robtarget Target_2170_2:=[[35.111,85.474,0],[0.726314069,0.009187373,0.687236181,-0.009481395],[-2,0,-1,0],[9E+09,9E+09,9E+09,9E+09,9E+09,9E+09]];
    CONST robtarget Target_2180_2:=[[40.922,85.474,0],[0.726314069,0.009187373,0.687236181,-0.009481395],[-2,0,-1,0],[9E+09,9E+09,9E+09,9E+09,9E+09,9E+09]];
    CONST robtarget Target_2190_2:=[[40.922,79.566,0],[0.726314069,0.009187373,0.687236181,-0.009481395],[-2,0,-1,0],[9E+09,9E+09,9E+09,9E+09,9E+09,9E+09]];
